LIN {X 0,Y 517.337,Z 394.066,A -85,B 0,C 180,E1 -4968.019,E2 -4968.019} C_VEL
LIN {X 0,Y 517.611,Z 384.123,A -85,B 0,C 180,E1 -4969.017,E2 -4969.017} C_VEL
LIN {X 0,Y 517.898,Z 374.015,A -85,B 0,C 180,E1 -4969.831,E2 -4969.831} C_VEL
LIN {X 0,Y 518.219,Z 361.881,A -85,B 0,C 180,E1 -4970.601,E2 -4970.601} C_VEL
LIN {X 0,Y 518.436,Z 350.506,A -85,B 0,C 180,E1 -4971.157,E2 -4971.157} C_VEL
LIN {X 0,Y 518.274,Z 345.949,A -85,B 0,C 180,E1 -4971.343,E2 -4971.343} C_VEL
LIN {X 0,Y 516.939,Z 341.096,A -85,B 0,C 180,E1 -4971.561,E2 -4971.561} C_VEL
LIN {X 0,Y 516.912,Z 341.099,A -85,B 0,C 180,E1 -4974.927,E2 -4974.927} C_VEL
LIN {X 0,Y 516.926,Z 341.098,A -85,B 0,C 180,E1 -4977.904,E2 -4977.904} C_VEL
LIN {X 0,Y 516.894,Z 341.103,A -85,B 0,C 180,E1 -4980.203,E2 -4980.203} C_VEL
LIN {X 0,Y 516.898,Z 341.101,A -85,B 0,C 180,E1 -4982.946,E2 -4982.946} C_VEL
LIN {X 0,Y 516.872,Z 341.104,A -85,B 0,C 180,E1 -4985.78,E2 -4985.78} C_VEL
LIN {X 0,Y 516.881,Z 341.103,A -85,B 0,C 180,E1 -4988.715,E2 -4988.715} C_VEL
LIN {X 0,Y 516.915,Z 341.097,A -85,B 0,C 180,E1 -4991.774,E2 -4991.774} C_VEL
LIN {X 0,Y 516.923,Z 341.097,A -85,B 0,C 180,E1 -4995.009,E2 -4995.009} C_VEL
LIN {X 0,Y 516.923,Z 341.099,A -85,B 0,C 180,E1 -4998.397,E2 -4998.397} C_VEL
LIN {X 0,Y 516.906,Z 341.1,A -85,B 0,C 180,E1 -5001.286,E2 -5001.286} C_VEL
LIN {X 0,Y 516.891,Z 341.1,A -85,B 0,C 180,E1 -5004.221,E2 -5004.221} C_VEL
LIN {X 0,Y 516.898,Z 341.099,A -85,B 0,C 180,E1 -5007.053,E2 -5007.053} C_VEL
LIN {X 0,Y 516.901,Z 341.087,A -85,B 0,C 180,E1 -5009.796,E2 -5009.796} C_VEL
LIN {X 0,Y 516.929,Z 341.095,A -85,B 0,C 180,E1 -5012.467,E2 -5012.467} C_VEL
LIN {X 0,Y 516.911,Z 341.098,A -85,B 0,C 180,E1 -5015.072,E2 -5015.072} C_VEL
LIN {X 0,Y 516.886,Z 341.103,A -85,B 0,C 180,E1 -5018.462,E2 -5018.462} C_VEL
LIN {X 0,Y 516.904,Z 341.098,A -85,B 0,C 180,E1 -5020.955,E2 -5020.955} C_VEL
LIN {X 0,Y 516.916,Z 341.098,A -85,B 0,C 180,E1 -5023.41,E2 -5023.41} C_VEL
LIN {X 0,Y 516.905,Z 341.099,A -85,B 0,C 180,E1 -5025.834,E2 -5025.834} C_VEL
LIN {X 0,Y 517.002,Z 341.088,A -85,B 0,C 180,E1 -5028.234,E2 -5028.234} C_VEL
LIN {X 0,Y 516.97,Z 341.092,A -85,B 0,C 180,E1 -5031.399,E2 -5031.399} C_VEL
LIN {X 0,Y 517.008,Z 341.083,A -85,B 0,C 180,E1 -5033.757,E2 -5033.757} C_VEL
LIN {X 0,Y 517.082,Z 341.077,A -85,B 0,C 180,E1 -5037.663,E2 -5037.663} C_VEL
LIN {X 0,Y 517.093,Z 341.074,A -85,B 0,C 180,E1 -5040.779,E2 -5040.779} C_VEL
LIN {X 0,Y 517.013,Z 341.087,A -85,B 0,C 180,E1 -5043.117,E2 -5043.117} C_VEL
LIN {X 0,Y 517.008,Z 341.086,A -85,B 0,C 180,E1 -5046.243,E2 -5046.243} C_VEL
LIN {X 0,Y 516.952,Z 341.091,A -85,B 0,C 180,E1 -5049.389,E2 -5049.389} C_VEL
LIN {X 0,Y 516.949,Z 341.093,A -85,B 0,C 180,E1 -5051.807,E2 -5051.807} C_VEL
LIN {X 0,Y 516.941,Z 341.095,A -85,B 0,C 180,E1 -5055.147,E2 -5055.147} C_VEL
LIN {X 0,Y 516.923,Z 341.097,A -85,B 0,C 180,E1 -5058.222,E2 -5058.222} C_VEL
LIN {X 0,Y 516.909,Z 341.097,A -85,B 0,C 180,E1 -5060.702,E2 -5060.702} C_VEL
LIN {X 0,Y 516.908,Z 341.099,A -85,B 0,C 180,E1 -5064.072,E2 -5064.072} C_VEL
LIN {X 0,Y 516.927,Z 341.097,A -85,B 0,C 180,E1 -5066.658,E2 -5066.658} C_VEL
LIN {X 0,Y 516.922,Z 341.098,A -85,B 0,C 180,E1 -5069.527,E2 -5069.527} C_VEL
LIN {X 0,Y 516.899,Z 341.1,A -85,B 0,C 180,E1 -5072.545,E2 -5072.545} C_VEL
LIN {X 0,Y 516.882,Z 341.102,A -85,B 0,C 180,E1 -5075.333,E2 -5075.333} C_VEL
LIN {X 0,Y 516.884,Z 341.102,A -85,B 0,C 180,E1 -5077.944,E2 -5077.944} C_VEL
LIN {X 0,Y 516.903,Z 341.099,A -85,B 0,C 180,E1 -5080.74,E2 -5080.74} C_VEL
LIN {X 0,Y 516.881,Z 341.102,A -85,B 0,C 180,E1 -5083.903,E2 -5083.903} C_VEL
LIN {X 0,Y 516.882,Z 341.101,A -85,B 0,C 180,E1 -5086.107,E2 -5086.107} C_VEL
LIN {X 0,Y 516.907,Z 341.102,A -85,B 0,C 180,E1 -5089.261,E2 -5089.261} C_VEL
LIN {X 0,Y 516.925,Z 341.244,A -85,B 0,C 180,E1 -5091.538,E2 -5091.538} C_VEL
LIN {X 0,Y 518.509,Z 349.549,A -85,B 0,C 180,E1 -5093.871,E2 -5093.871} C_VEL
LIN {X 0,Y 518.338,Z 357.102,A -85,B 0,C 180,E1 -5095.8,E2 -5095.8} C_VEL
LIN {X 0,Y 517.884,Z 371.915,A -85,B 0,C 180,E1 -5099.41,E2 -5099.41} C_VEL
LIN {X 0,Y 517.599,Z 385.199,A -85,B 0,C 180,E1 -5102.507,E2 -5102.507} C_VEL
LIN {X 0,Y 517.364,Z 398.58,A -85,B 0,C 180,E1 -5105.526,E2 -5105.526} C_VEL
LIN {X 0,Y 517.164,Z 411.994,A -85,B 0,C 180,E1 -5108.475,E2 -5108.475} C_VEL
LIN {X 0,Y 516.997,Z 423.426,A -85,B 0,C 180,E1 -5110.959,E2 -5110.959} C_VEL
LIN {X 0,Y 516.858,Z 435.03,A -85,B 0,C 180,E1 -5113.409,E2 -5113.409} C_VEL
LIN {X 0,Y 516.733,Z 447.489,A -85,B 0,C 180,E1 -5116.056,E2 -5116.056} C_VEL
LIN {X 0,Y 518.309,Z 459.336,A -85,B 0,C 180,E1 -5116.349,E2 -5116.349} C_VEL
LIN {X 0,Y 518.198,Z 472.484,A -85,B 0,C 180,E1 -5116.77,E2 -5116.77} C_VEL
LIN {X 0,Y 517.966,Z 483.611,A -85,B 0,C 180,E1 -5117.263,E2 -5117.263} C_VEL
LIN {X 0,Y 517.668,Z 495.877,A -85,B 0,C 180,E1 -5117.972,E2 -5117.972} C_VEL
LIN {X 0,Y 517.351,Z 507.545,A -85,B 0,C 180,E1 -5118.839,E2 -5118.839} C_VEL
LIN {X 0,Y 517.042,Z 518.18,A -85,B 0,C 180,E1 -5119.823,E2 -5119.823} C_VEL
LIN {X 0,Y 516.815,Z 526.807,A -85,B 0,C 180,E1 -5120.806,E2 -5120.806} C_VEL
LIN {X 0,Y 516.616,Z 535.236,A -85,B 0,C 180,E1 -5121.985,E2 -5121.985} C_VEL
LIN {X 0,Y 516.48,Z 542.24,A -85,B 0,C 180,E1 -5123.2,E2 -5123.2} C_VEL
LIN {X 0,Y 516.405,Z 548.283,A -85,B 0,C 180,E1 -5124.534,E2 -5124.534} C_VEL
LIN {X 0,Y 516.36,Z 552.34,A -85,B 0,C 180,E1 -5125.707,E2 -5125.707} C_VEL
LIN {X 0,Y 516.282,Z 555.331,A -85,B 0,C 180,E1 -5126.879,E2 -5126.879} C_VEL
LIN {X 0,Y 516.261,Z 556.758,A -85,B 0,C 180,E1 -5127.66,E2 -5127.66} C_VEL
LIN {X 0,Y 516.161,Z 558.388,A -85,B 0,C 180,E1 -5129.22,E2 -5129.22} C_VEL
LIN {X 0,Y 516.158,Z 558.609,A -85,B 0,C 180,E1 -5130.001,E2 -5130.001} C_VEL
LIN {X 0,Y 516.161,Z 558.388,A -85,B 0,C 180,E1 -5130.781,E2 -5130.781} C_VEL
LIN {X 0,Y 516.261,Z 556.761,A -85,B 0,C 180,E1 -5132.341,E2 -5132.341} C_VEL
LIN {X 0,Y 516.282,Z 555.335,A -85,B 0,C 180,E1 -5133.122,E2 -5133.122} C_VEL
LIN {X 0,Y 516.343,Z 552.34,A -85,B 0,C 180,E1 -5134.294,E2 -5134.294} C_VEL
LIN {X 0,Y 516.405,Z 548.284,A -85,B 0,C 180,E1 -5135.467,E2 -5135.467} C_VEL
LIN {X 0,Y 516.481,Z 542.255,A -85,B 0,C 180,E1 -5136.799,E2 -5136.799} C_VEL
LIN {X 0,Y 516.617,Z 535.245,A -85,B 0,C 180,E1 -5138.016,E2 -5138.016} C_VEL
LIN {X 0,Y 516.816,Z 526.82,A -85,B 0,C 180,E1 -5139.195,E2 -5139.195} C_VEL
LIN {X 0,Y 517.038,Z 518.196,A -85,B 0,C 180,E1 -5140.179,E2 -5140.179} C_VEL
LIN {X 0,Y 517.39,Z 507.571,A -85,B 0,C 180,E1 -5141.162,E2 -5141.162} C_VEL
LIN {X 0,Y 517.627,Z 496.24,A -85,B 0,C 180,E1 -5142.007,E2 -5142.007} C_VEL
LIN {X 0,Y 517.95,Z 485.582,A -85,B 0,C 180,E1 -5142.639,E2 -5142.639} C_VEL
LIN {X 0,Y 518.174,Z 473.805,A -85,B 0,C 180,E1 -5143.182,E2 -5143.182} C_VEL
LIN {X 0,Y 518.435,Z 460.279,A -85,B 0,C 180,E1 -5143.624,E2 -5143.624} C_VEL
LIN {X 0,Y 516.87,Z 449.371,A -85,B 0,C 180,E1 -5143.898,E2 -5143.898} C_VEL
LIN {X 0,Y 516.731,Z 447.432,A -85,B 0,C 180,E1 -5143.971,E2 -5143.971} C_VEL
LIN {X 0,Y 516.937,Z 433.234,A -85,B 0,C 180,E1 -5146.996,E2 -5146.996} C_VEL
LIN {X 0,Y 517.111,Z 417.675,A -85,B 0,C 180,E1 -5150.319,E2 -5150.319} C_VEL
LIN {X 0,Y 517.307,Z 404.507,A -85,B 0,C 180,E1 -5153.203,E2 -5153.203} C_VEL
LIN {X 0,Y 517.52,Z 390.545,A -85,B 0,C 180,E1 -5156.325,E2 -5156.325} C_VEL
LIN {X 0,Y 517.743,Z 377.723,A -85,B 0,C 180,E1 -5159.254,E2 -5159.254} C_VEL
LIN {X 0,Y 518.003,Z 366.207,A -85,B 0,C 180,E1 -5161.947,E2 -5161.947} C_VEL
LIN {X 0,Y 518.417,Z 352.975,A -85,B 0,C 180,E1 -5165.141,E2 -5165.141} C_VEL
LIN {X 0,Y 518.322,Z 348.977,A -85,B 0,C 180,E1 -5166.145,E2 -5166.145} C_VEL
LIN {X 0,Y 516.879,Z 341.103,A -85,B 0,C 180,E1 -5168.305,E2 -5168.305} C_VEL
LIN {X 0,Y 516.921,Z 341.098,A -85,B 0,C 180,E1 -5171.602,E2 -5171.602} C_VEL
LIN {X 0,Y 516.928,Z 341.098,A -85,B 0,C 180,E1 -5175.01,E2 -5175.01} C_VEL
LIN {X 0,Y 516.92,Z 341.098,A -85,B 0,C 180,E1 -5178.399,E2 -5178.399} C_VEL
LIN {X 0,Y 516.888,Z 341.101,A -85,B 0,C 180,E1 -5181.285,E2 -5181.285} C_VEL
LIN {X 0,Y 516.876,Z 341.103,A -85,B 0,C 180,E1 -5184.22,E2 -5184.22} C_VEL
LIN {X 0,Y 516.902,Z 341.1,A -85,B 0,C 180,E1 -5187.054,E2 -5187.054} C_VEL
LIN {X 0,Y 516.898,Z 341.1,A -85,B 0,C 180,E1 -5189.797,E2 -5189.797} C_VEL
LIN {X 0,Y 516.931,Z 341.095,A -85,B 0,C 180,E1 -5192.468,E2 -5192.468} C_VEL
LIN {X 0,Y 516.916,Z 341.099,A -85,B 0,C 180,E1 -5195.072,E2 -5195.072} C_VEL
LIN {X 0,Y 516.876,Z 341.102,A -85,B 0,C 180,E1 -5197.622,E2 -5197.622} C_VEL
LIN {X 0,Y 516.937,Z 341.095,A -85,B 0,C 180,E1 -5200.13,E2 -5200.13} C_VEL
LIN {X 0,Y 516.913,Z 341.098,A -85,B 0,C 180,E1 -5202.596,E2 -5202.596} C_VEL
LIN {X 0,Y 516.948,Z 341.094,A -85,B 0,C 180,E1 -5205.03,E2 -5205.03} C_VEL
LIN {X 0,Y 516.972,Z 341.091,A -85,B 0,C 180,E1 -5208.234,E2 -5208.234} C_VEL
LIN {X 0,Y 516.972,Z 341.089,A -85,B 0,C 180,E1 -5211.4,E2 -5211.4} C_VEL
LIN {X 0,Y 517.016,Z 341.084,A -85,B 0,C 180,E1 -5213.757,E2 -5213.757} C_VEL
LIN {X 0,Y 517.087,Z 341.077,A -85,B 0,C 180,E1 -5217.663,E2 -5217.663} C_VEL
LIN {X 0,Y 517.101,Z 341.075,A -85,B 0,C 180,E1 -5220.779,E2 -5220.779} C_VEL
LIN {X 0,Y 517.018,Z 341.085,A -85,B 0,C 180,E1 -5223.117,E2 -5223.117} C_VEL
LIN {X 0,Y 517.015,Z 341.086,A -85,B 0,C 180,E1 -5226.243,E2 -5226.243} C_VEL
LIN {X 0,Y 516.961,Z 341.091,A -85,B 0,C 180,E1 -5229.389,E2 -5229.389} C_VEL
LIN {X 0,Y 516.959,Z 341.092,A -85,B 0,C 180,E1 -5231.807,E2 -5231.807} C_VEL
LIN {X 0,Y 516.951,Z 341.092,A -85,B 0,C 180,E1 -5235.147,E2 -5235.147} C_VEL
LIN {X 0,Y 516.932,Z 341.095,A -85,B 0,C 180,E1 -5238.222,E2 -5238.222} C_VEL
LIN {X 0,Y 516.919,Z 341.096,A -85,B 0,C 180,E1 -5240.702,E2 -5240.702} C_VEL
LIN {X 0,Y 516.918,Z 341.097,A -85,B 0,C 180,E1 -5244.072,E2 -5244.072} C_VEL
LIN {X 0,Y 516.932,Z 341.096,A -85,B 0,C 180,E1 -5246.658,E2 -5246.658} C_VEL
LIN {X 0,Y 516.917,Z 341.098,A -85,B 0,C 180,E1 -5249.524,E2 -5249.524} C_VEL
LIN {X 0,Y 516.904,Z 341.099,A -85,B 0,C 180,E1 -5252.544,E2 -5252.544} C_VEL
LIN {X 0,Y 516.873,Z 341.103,A -85,B 0,C 180,E1 -5255.33,E2 -5255.33} C_VEL
LIN {X 0,Y 516.888,Z 341.102,A -85,B 0,C 180,E1 -5257.943,E2 -5257.943} C_VEL
LIN {X 0,Y 516.891,Z 341.1,A -85,B 0,C 180,E1 -5260.741,E2 -5260.741} C_VEL
LIN {X 0,Y 516.889,Z 341.101,A -85,B 0,C 180,E1 -5262.831,E2 -5262.831} C_VEL
LIN {X 0,Y 516.93,Z 341.097,A -85,B 0,C 180,E1 -5265.01,E2 -5265.01} C_VEL
LIN {X 0,Y 516.923,Z 341.097,A -85,B 0,C 180,E1 -5268.398,E2 -5268.398} C_VEL
LIN {X 0,Y 516.888,Z 341.101,A -85,B 0,C 180,E1 -5270.301,E2 -5270.301} C_VEL
LIN {X 0,Y 516.213,Z 341.185,A -85,B 0,C 180,E1 -5270.951,E2 -5270.951} C_VEL
LIN {X 0,Y 513.355,Z 341.544,A -85,B 0,C 180,E1 -5272.006,E2 -5272.006} C_VEL
LIN {X 0,Y 510.94,Z 341.846,A -85,B 0,C 180,E1 -5272.857,E2 -5272.857} C_VEL
LIN {X 0,Y 509.9,Z 341.974,A -85,B 0,C 180,E1 -5273.513,E2 -5273.513} C_VEL
LIN {X 0,Y 509.813,Z 341.983,A -85,B 0,C 180,E1 -5273.736,E2 -5273.736} C_VEL
LIN {X 0,Y 509.866,Z 341.975,A -85,B 0,C 180,E1 -5276.539,E2 -5276.539} C_VEL
LIN {X 0,Y 509.85,Z 341.979,A -85,B 0,C 180,E1 -5279.334,E2 -5279.334} C_VEL
LIN {X 0,Y 509.897,Z 341.97,A -85,B 0,C 180,E1 -5282.054,E2 -5282.054} C_VEL
LIN {X 0,Y 509.884,Z 341.974,A -85,B 0,C 180,E1 -5284.704,E2 -5284.704} C_VEL
LIN {X 0,Y 509.834,Z 341.979,A -85,B 0,C 180,E1 -5287.458,E2 -5287.458} C_VEL
LIN {X 0,Y 509.924,Z 341.967,A -85,B 0,C 180,E1 -5289.844,E2 -5289.844} C_VEL
LIN {X 0,Y 509.889,Z 341.972,A -85,B 0,C 180,E1 -5293.174,E2 -5293.174} C_VEL
LIN {X 0,Y 509.871,Z 341.973,A -85,B 0,C 180,E1 -5295.634,E2 -5295.634} C_VEL
LIN {X 0,Y 509.921,Z 341.969,A -85,B 0,C 180,E1 -5298.874,E2 -5298.874} C_VEL
LIN {X 0,Y 509.959,Z 341.964,A -85,B 0,C 180,E1 -5302.078,E2 -5302.078} C_VEL
LIN {X 0,Y 509.974,Z 341.963,A -85,B 0,C 180,E1 -5304.34,E2 -5304.34} C_VEL
LIN {X 0,Y 511.619,Z 348.18,A -85,B 0,C 180,E1 -5304.63,E2 -5304.63} C_VEL
LIN {X 0,Y 511.412,Z 359.998,A -85,B 0,C 180,E1 -5305.171,E2 -5305.171} C_VEL
LIN {X 0,Y 511.143,Z 371.42,A -85,B 0,C 180,E1 -5305.86,E2 -5305.86} C_VEL
LIN {X 0,Y 510.795,Z 382.869,A -85,B 0,C 180,E1 -5306.746,E2 -5306.746} C_VEL
LIN {X 0,Y 510.5,Z 392.107,A -85,B 0,C 180,E1 -5307.632,E2 -5307.632} C_VEL
LIN {X 0,Y 510.193,Z 400.557,A -85,B 0,C 180,E1 -5308.618,E2 -5308.618} C_VEL
LIN {X 0,Y 509.931,Z 408.768,A -85,B 0,C 180,E1 -5309.802,E2 -5309.802} C_VEL
LIN {X 0,Y 509.631,Z 416.37,A -85,B 0,C 180,E1 -5311.185,E2 -5311.185} C_VEL
LIN {X 0,Y 509.497,Z 421.464,A -85,B 0,C 180,E1 -5312.371,E2 -5312.371} C_VEL
LIN {X 0,Y 509.46,Z 425.423,A -85,B 0,C 180,E1 -5313.558,E2 -5313.558} C_VEL
LIN {X 0,Y 509.347,Z 428.382,A -85,B 0,C 180,E1 -5314.748,E2 -5314.748} C_VEL
LIN {X 0,Y 509.37,Z 429.832,A -85,B 0,C 180,E1 -5315.542,E2 -5315.542} C_VEL
LIN {X 0,Y 509.331,Z 431.496,A -85,B 0,C 180,E1 -5317.133,E2 -5317.133} C_VEL
LIN {X 0,Y 509.334,Z 431.764,A -85,B 0,C 180,E1 -5317.931,E2 -5317.931} C_VEL
LIN {X 0,Y 509.303,Z 431.64,A -85,B 0,C 180,E1 -5318.73,E2 -5318.73} C_VEL
LIN {X 0,Y 509.29,Z 430.153,A -85,B 0,C 180,E1 -5320.334,E2 -5320.334} C_VEL
LIN {X 0,Y 509.393,Z 427.838,A -85,B 0,C 180,E1 -5321.598,E2 -5321.598} C_VEL
LIN {X 0,Y 509.441,Z 424.792,A -85,B 0,C 180,E1 -5322.751,E2 -5322.751} C_VEL
LIN {X 0,Y 509.555,Z 420.523,A -85,B 0,C 180,E1 -5323.967,E2 -5323.967} C_VEL
LIN {X 0,Y 509.743,Z 415.022,A -85,B 0,C 180,E1 -5325.186,E2 -5325.186} C_VEL
LIN {X 0,Y 509.929,Z 408.09,A -85,B 0,C 180,E1 -5326.411,E2 -5326.411} C_VEL
LIN {X 0,Y 510.241,Z 399.294,A -85,B 0,C 180,E1 -5327.639,E2 -5327.639} C_VEL
LIN {X 0,Y 510.571,Z 390.201,A -85,B 0,C 180,E1 -5328.664,E2 -5328.664} C_VEL
LIN {X 0,Y 510.846,Z 380.073,A -85,B 0,C 180,E1 -5329.593,E2 -5329.593} C_VEL
LIN {X 0,Y 511.197,Z 369.49,A -85,B 0,C 180,E1 -5330.364,E2 -5330.364} C_VEL
LIN {X 0,Y 511.481,Z 357.788,A -85,B 0,C 180,E1 -5331.036,E2 -5331.036} C_VEL
LIN {X 0,Y 511.617,Z 348.497,A -85,B 0,C 180,E1 -5331.453,E2 -5331.453} C_VEL
LIN {X 0,Y 509.877,Z 341.975,A -85,B 0,C 180,E1 -5331.768,E2 -5331.768} C_VEL
LIN {X 0,Y 509.879,Z 341.975,A -85,B 0,C 180,E1 -5335.295,E2 -5335.295} C_VEL
LIN {X 0,Y 509.898,Z 341.973,A -85,B 0,C 180,E1 -5338.1,E2 -5338.1} C_VEL
LIN {X 0,Y 509.848,Z 341.978,A -85,B 0,C 180,E1 -5341.279,E2 -5341.279} C_VEL
LIN {X 0,Y 509.858,Z 341.976,A -85,B 0,C 180,E1 -5344.202,E2 -5344.202} C_VEL
LIN {X 0,Y 509.817,Z 341.984,A -85,B 0,C 180,E1 -5347.34,E2 -5347.34} C_VEL
LIN {X 0,Y 509.839,Z 341.98,A -85,B 0,C 180,E1 -5350.381,E2 -5350.381} C_VEL
LIN {X 0,Y 509.84,Z 341.979,A -85,B 0,C 180,E1 -5353.064,E2 -5353.064} C_VEL
LIN {X 0,Y 509.831,Z 341.981,A -85,B 0,C 180,E1 -5355.792,E2 -5355.792} C_VEL
LIN {X 0,Y 509.865,Z 341.978,A -85,B 0,C 180,E1 -5358.575,E2 -5358.575} C_VEL
LIN {X 0,Y 509.859,Z 341.978,A -85,B 0,C 180,E1 -5361.662,E2 -5361.662} C_VEL
LIN {X 0,Y 509.847,Z 341.979,A -85,B 0,C 180,E1 -5364.623,E2 -5364.623} C_VEL
LIN {X 0,Y 509.866,Z 341.974,A -85,B 0,C 180,E1 -5367.481,E2 -5367.481} C_VEL
LIN {X 0,Y 509.88,Z 341.962,A -85,B 0,C 180,E1 -5370.268,E2 -5370.268} C_VEL
LIN {X 0,Y 509.886,Z 341.971,A -85,B 0,C 180,E1 -5372.944,E2 -5372.944} C_VEL
LIN {X 0,Y 509.869,Z 341.974,A -85,B 0,C 180,E1 -5375.574,E2 -5375.574} C_VEL
LIN {X 0,Y 509.821,Z 341.98,A -85,B 0,C 180,E1 -5378.148,E2 -5378.148} C_VEL
LIN {X 0,Y 509.864,Z 341.975,A -85,B 0,C 180,E1 -5380.681,E2 -5380.681} C_VEL
LIN {X 0,Y 509.886,Z 341.971,A -85,B 0,C 180,E1 -5383.175,E2 -5383.175} C_VEL
LIN {X 0,Y 509.872,Z 341.975,A -85,B 0,C 180,E1 -5385.634,E2 -5385.634} C_VEL
LIN {X 0,Y 509.929,Z 341.968,A -85,B 0,C 180,E1 -5388.875,E2 -5388.875} C_VEL
LIN {X 0,Y 509.95,Z 341.966,A -85,B 0,C 180,E1 -5392.078,E2 -5392.078} C_VEL
LIN {X 0,Y 509.981,Z 341.959,A -85,B 0,C 180,E1 -5394.464,E2 -5394.464} C_VEL
LIN {X 0,Y 510.053,Z 341.952,A -85,B 0,C 180,E1 -5397.631,E2 -5397.631} C_VEL
LIN {X 0,Y 510.063,Z 341.949,A -85,B 0,C 180,E1 -5400.789,E2 -5400.789} C_VEL
LIN {X 0,Y 509.955,Z 341.966,A -85,B 0,C 180,E1 -5403.16,E2 -5403.16} C_VEL
LIN {X 0,Y 509.976,Z 341.963,A -85,B 0,C 180,E1 -5406.329,E2 -5406.329} C_VEL
LIN {X 0,Y 509.914,Z 341.969,A -85,B 0,C 180,E1 -5408.72,E2 -5408.72} C_VEL
LIN {X 0,Y 509.901,Z 341.971,A -85,B 0,C 180,E1 -5411.932,E2 -5411.932} C_VEL
LIN {X 0,Y 509.89,Z 341.974,A -85,B 0,C 180,E1 -5415.242,E2 -5415.242} C_VEL
LIN {X 0,Y 509.885,Z 341.972,A -85,B 0,C 180,E1 -5418.001,E2 -5418.001} C_VEL
LIN {X 0,Y 509.847,Z 341.977,A -85,B 0,C 180,E1 -5421.002,E2 -5421.002} C_VEL
LIN {X 0,Y 509.834,Z 341.979,A -85,B 0,C 180,E1 -5423.563,E2 -5423.563} C_VEL
LIN {X 0,Y 509.911,Z 341.972,A -85,B 0,C 180,E1 -5426.379,E2 -5426.379} C_VEL
LIN {X 0,Y 509.883,Z 341.975,A -85,B 0,C 180,E1 -5428.844,E2 -5428.844} C_VEL
LIN {X 0,Y 509.824,Z 341.982,A -85,B 0,C 180,E1 -5431.59,E2 -5431.59} C_VEL
LIN {X 0,Y 509.852,Z 341.978,A -85,B 0,C 180,E1 -5434.413,E2 -5434.413} C_VEL
LIN {X 0,Y 509.821,Z 341.982,A -85,B 0,C 180,E1 -5437.341,E2 -5437.341} C_VEL
LIN {X 0,Y 509.86,Z 341.977,A -85,B 0,C 180,E1 -5440.38,E2 -5440.38} C_VEL
LIN {X 0,Y 509.838,Z 341.981,A -85,B 0,C 180,E1 -5443.065,E2 -5443.065} C_VEL
LIN {X 0,Y 509.83,Z 341.981,A -85,B 0,C 180,E1 -5445.793,E2 -5445.793} C_VEL
LIN {X 0,Y 509.87,Z 341.977,A -85,B 0,C 180,E1 -5448.577,E2 -5448.577} C_VEL
LIN {X 0,Y 509.906,Z 342.094,A -85,B 0,C 180,E1 -5451.258,E2 -5451.258} C_VEL
LIN {X 0,Y 511.562,Z 350.947,A -85,B 0,C 180,E1 -5453.791,E2 -5453.791} C_VEL
LIN {X 0,Y 511.394,Z 358.315,A -85,B 0,C 180,E1 -5455.706,E2 -5455.706} C_VEL
LIN {X 0,Y 510.939,Z 371.404,A -85,B 0,C 180,E1 -5458.959,E2 -5458.959} C_VEL
LIN {X 0,Y 510.599,Z 384.561,A -85,B 0,C 180,E1 -5462.097,E2 -5462.097} C_VEL
LIN {X 0,Y 510.365,Z 397.528,A -85,B 0,C 180,E1 -5465.088,E2 -5465.088} C_VEL
LIN {X 0,Y 510.12,Z 411.233,A -85,B 0,C 180,E1 -5468.163,E2 -5468.163} C_VEL
LIN {X 0,Y 509.933,Z 422.681,A -85,B 0,C 180,E1 -5470.685,E2 -5470.685} C_VEL
LIN {X 0,Y 509.793,Z 434.11,A -85,B 0,C 180,E1 -5473.172,E2 -5473.172} C_VEL
LIN {X 0,Y 509.66,Z 446.577,A -85,B 0,C 180,E1 -5475.858,E2 -5475.858} C_VEL
LIN {X 0,Y 511.033,Z 457.931,A -85,B 0,C 180,E1 -5476.138,E2 -5476.138} C_VEL
LIN {X 0,Y 511.475,Z 462.135,A -85,B 0,C 180,E1 -5476.264,E2 -5476.264} C_VEL
LIN {X 0,Y 511.177,Z 475.257,A -85,B 0,C 180,E1 -5476.737,E2 -5476.737} C_VEL
LIN {X 0,Y 510.84,Z 487.929,A -85,B 0,C 180,E1 -5477.369,E2 -5477.369} C_VEL
LIN {X 0,Y 510.567,Z 499.026,A -85,B 0,C 180,E1 -5478.085,E2 -5478.085} C_VEL
LIN {X 0,Y 510.21,Z 510.079,A -85,B 0,C 180,E1 -5478.982,E2 -5478.982} C_VEL
LIN {X 0,Y 509.927,Z 519.109,A -85,B 0,C 180,E1 -5479.88,E2 -5479.88} C_VEL
LIN {X 0,Y 509.68,Z 528.943,A -85,B 0,C 180,E1 -5481.076,E2 -5481.076} C_VEL
LIN {X 0,Y 509.512,Z 536.792,A -85,B 0,C 180,E1 -5482.272,E2 -5482.272} C_VEL
LIN {X 0,Y 509.341,Z 544.029,A -85,B 0,C 180,E1 -5483.663,E2 -5483.663} C_VEL
LIN {X 0,Y 509.255,Z 548.853,A -85,B 0,C 180,E1 -5484.854,E2 -5484.854} C_VEL
LIN {X 0,Y 509.303,Z 552.555,A -85,B 0,C 180,E1 -5486.044,E2 -5486.044} C_VEL
LIN {X 0,Y 509.232,Z 554.454,A -85,B 0,C 180,E1 -5486.836,E2 -5486.836} C_VEL
LIN {X 0,Y 509.206,Z 555.882,A -85,B 0,C 180,E1 -5487.628,E2 -5487.628} C_VEL
LIN {X 0,Y 509.114,Z 557.515,A -85,B 0,C 180,E1 -5489.21,E2 -5489.21} C_VEL
LIN {X 0,Y 509.112,Z 557.738,A -85,B 0,C 180,E1 -5490.001,E2 -5490.001} C_VEL
LIN {X 0,Y 509.114,Z 557.517,A -85,B 0,C 180,E1 -5490.792,E2 -5490.792} C_VEL
LIN {X 0,Y 509.205,Z 555.89,A -85,B 0,C 180,E1 -5492.374,E2 -5492.374} C_VEL
LIN {X 0,Y 509.232,Z 554.465,A -85,B 0,C 180,E1 -5493.165,E2 -5493.165} C_VEL
LIN {X 0,Y 509.269,Z 551.466,A -85,B 0,C 180,E1 -5494.354,E2 -5494.354} C_VEL
LIN {X 0,Y 509.344,Z 547.412,A -85,B 0,C 180,E1 -5495.543,E2 -5495.543} C_VEL
LIN {X 0,Y 509.403,Z 541.634,A -85,B 0,C 180,E1 -5496.845,E2 -5496.845} C_VEL
LIN {X 0,Y 509.563,Z 534.37,A -85,B 0,C 180,E1 -5498.128,E2 -5498.128} C_VEL
LIN {X 0,Y 509.759,Z 525.944,A -85,B 0,C 180,E1 -5499.323,E2 -5499.323} C_VEL
LIN {X 0,Y 510.006,Z 517.32,A -85,B 0,C 180,E1 -5500.32,E2 -5500.32} C_VEL
LIN {X 0,Y 510.353,Z 506.691,A -85,B 0,C 180,E1 -5501.317,E2 -5501.317} C_VEL
LIN {X 0,Y 510.616,Z 495.361,A -85,B 0,C 180,E1 -5502.174,E2 -5502.174} C_VEL
LIN {X 0,Y 510.959,Z 484.704,A -85,B 0,C 180,E1 -5502.815,E2 -5502.815} C_VEL
LIN {X 0,Y 511.239,Z 472.931,A -85,B 0,C 180,E1 -5503.364,E2 -5503.364} C_VEL
LIN {X 0,Y 511.36,Z 460.306,A -85,B 0,C 180,E1 -5503.791,E2 -5503.791} C_VEL
LIN {X 0,Y 509.739,Z 448.093,A -85,B 0,C 180,E1 -5504.103,E2 -5504.103} C_VEL
LIN {X 0,Y 509.676,Z 446.545,A -85,B 0,C 180,E1 -5504.168,E2 -5504.168} C_VEL
LIN {X 0,Y 509.89,Z 430.427,A -85,B 0,C 180,E1 -5507.653,E2 -5507.653} C_VEL
LIN {X 0,Y 510.045,Z 416.632,A -85,B 0,C 180,E1 -5510.676,E2 -5510.676} C_VEL
LIN {X 0,Y 510.269,Z 403.803,A -85,B 0,C 180,E1 -5513.543,E2 -5513.543} C_VEL
LIN {X 0,Y 510.493,Z 390.743,A -85,B 0,C 180,E1 -5516.509,E2 -5516.509} C_VEL
LIN {X 0,Y 510.791,Z 377.023,A -85,B 0,C 180,E1 -5519.692,E2 -5519.692} C_VEL
LIN {X 0,Y 511.079,Z 364.376,A -85,B 0,C 180,E1 -5522.709,E2 -5522.709} C_VEL
LIN {X 0,Y 511.487,Z 352.891,A -85,B 0,C 180,E1 -5525.539,E2 -5525.539} C_VEL
LIN {X 0,Y 511.122,Z 348.652,A -85,B 0,C 180,E1 -5526.643,E2 -5526.643} C_VEL
LIN {X 0,Y 509.852,Z 341.979,A -85,B 0,C 180,E1 -5528.465,E2 -5528.465} C_VEL
LIN {X 0,Y 509.862,Z 341.977,A -85,B 0,C 180,E1 -5531.426,E2 -5531.426} C_VEL
LIN {X 0,Y 509.862,Z 341.978,A -85,B 0,C 180,E1 -5534.668,E2 -5534.668} C_VEL
LIN {X 0,Y 509.861,Z 341.975,A -85,B 0,C 180,E1 -5538.104,E2 -5538.104} C_VEL
LIN {X 0,Y 509.853,Z 341.978,A -85,B 0,C 180,E1 -5540.648,E2 -5540.648} C_VEL
LIN {X 0,Y 509.83,Z 341.98,A -85,B 0,C 180,E1 -5543.647,E2 -5543.647} C_VEL
LIN {X 0,Y 509.865,Z 341.977,A -85,B 0,C 180,E1 -5546.54,E2 -5546.54} C_VEL
LIN {X 0,Y 509.852,Z 341.978,A -85,B 0,C 180,E1 -5549.335,E2 -5549.335} C_VEL
LIN {X 0,Y 509.897,Z 341.972,A -85,B 0,C 180,E1 -5552.055,E2 -5552.055} C_VEL
LIN {X 0,Y 509.882,Z 341.974,A -85,B 0,C 180,E1 -5554.704,E2 -5554.704} C_VEL
LIN {X 0,Y 509.862,Z 341.976,A -85,B 0,C 180,E1 -5557.45,E2 -5557.45} C_VEL
LIN {X 0,Y 509.922,Z 341.969,A -85,B 0,C 180,E1 -5559.845,E2 -5559.845} C_VEL
LIN {X 0,Y 509.881,Z 341.974,A -85,B 0,C 180,E1 -5563.175,E2 -5563.175} C_VEL
LIN {X 0,Y 509.87,Z 341.975,A -85,B 0,C 180,E1 -5565.634,E2 -5565.634} C_VEL
LIN {X 0,Y 509.918,Z 341.969,A -85,B 0,C 180,E1 -5568.875,E2 -5568.875} C_VEL
LIN {X 0,Y 509.957,Z 341.966,A -85,B 0,C 180,E1 -5572.079,E2 -5572.079} C_VEL
LIN {X 0,Y 509.988,Z 341.961,A -85,B 0,C 180,E1 -5574.465,E2 -5574.465} C_VEL
LIN {X 0,Y 510.058,Z 341.952,A -85,B 0,C 180,E1 -5577.631,E2 -5577.631} C_VEL
LIN {X 0,Y 510.071,Z 341.951,A -85,B 0,C 180,E1 -5580.79,E2 -5580.79} C_VEL
LIN {X 0,Y 509.96,Z 341.964,A -85,B 0,C 180,E1 -5583.16,E2 -5583.16} C_VEL
LIN {X 0,Y 509.984,Z 341.962,A -85,B 0,C 180,E1 -5586.33,E2 -5586.33} C_VEL
LIN {X 0,Y 509.923,Z 341.969,A -85,B 0,C 180,E1 -5588.72,E2 -5588.72} C_VEL
LIN {X 0,Y 509.911,Z 341.971,A -85,B 0,C 180,E1 -5591.932,E2 -5591.932} C_VEL
LIN {X 0,Y 509.901,Z 341.97,A -85,B 0,C 180,E1 -5595.242,E2 -5595.242} C_VEL
LIN {X 0,Y 509.895,Z 341.973,A -85,B 0,C 180,E1 -5598.001,E2 -5598.001} C_VEL
LIN {X 0,Y 509.857,Z 341.976,A -85,B 0,C 180,E1 -5601.002,E2 -5601.002} C_VEL
LIN {X 0,Y 509.877,Z 341.975,A -85,B 0,C 180,E1 -5604.426,E2 -5604.426} C_VEL
LIN {X 0,Y 509.891,Z 341.973,A -85,B 0,C 180,E1 -5607.056,E2 -5607.056} C_VEL
LIN {X 0,Y 509.864,Z 341.976,A -85,B 0,C 180,E1 -5609.751,E2 -5609.751} C_VEL
LIN {X 0,Y 509.881,Z 341.973,A -85,B 0,C 180,E1 -5612.774,E2 -5612.774} C_VEL
LIN {X 0,Y 509.833,Z 341.981,A -85,B 0,C 180,E1 -5615.578,E2 -5615.578} C_VEL
LIN {X 0,Y 509.858,Z 341.975,A -85,B 0,C 180,E1 -5618.338,E2 -5618.338} C_VEL
LIN {X 0,Y 509.864,Z 341.978,A -85,B 0,C 180,E1 -5621.425,E2 -5621.425} C_VEL
LIN {X 0,Y 509.864,Z 341.976,A -85,B 0,C 180,E1 -5624.668,E2 -5624.668} C_VEL
LIN {X 0,Y 509.865,Z 341.976,A -85,B 0,C 180,E1 -5628.103,E2 -5628.103} C_VEL
LIN {X 0,Y 509.852,Z 341.978,A -85,B 0,C 180,E1 -5630.647,E2 -5630.647} C_VEL
LIN {X 0,Y 509.813,Z 341.983,A -85,B 0,C 180,E1 -5633.736,E2 -5633.736} C_VEL
LIN {X 0,Y 509.154,Z 342.063,A -85,B 0,C 180,E1 -5634.395,E2 -5634.395} C_VEL
LIN {X 0,Y 506.347,Z 342.414,A -85,B 0,C 180,E1 -5635.468,E2 -5635.468} C_VEL
LIN {X 0,Y 503.96,Z 342.713,A -85,B 0,C 180,E1 -5636.331,E2 -5636.331} C_VEL
LIN {X 0,Y 502.913,Z 342.843,A -85,B 0,C 180,E1 -5636.998,E2 -5636.998} C_VEL
LIN {X 0,Y 502.815,Z 342.853,A -85,B 0,C 180,E1 -5637.223,E2 -5637.223} C_VEL
LIN {X 0,Y 502.821,Z 342.852,A -85,B 0,C 180,E1 -5640.065,E2 -5640.065} C_VEL
LIN {X 0,Y 502.838,Z 342.851,A -85,B 0,C 180,E1 -5642.533,E2 -5642.533} C_VEL
LIN {X 0,Y 502.834,Z 342.851,A -85,B 0,C 180,E1 -5645.299,E2 -5645.299} C_VEL
LIN {X 0,Y 502.787,Z 342.856,A -85,B 0,C 180,E1 -5647.826,E2 -5647.826} C_VEL
LIN {X 0,Y 502.832,Z 342.852,A -85,B 0,C 180,E1 -5650.4,E2 -5650.4} C_VEL
LIN {X 0,Y 502.837,Z 342.852,A -85,B 0,C 180,E1 -5652.931,E2 -5652.931} C_VEL
LIN {X 0,Y 502.852,Z 342.848,A -85,B 0,C 180,E1 -5655.429,E2 -5655.429} C_VEL
LIN {X 0,Y 502.885,Z 342.846,A -85,B 0,C 180,E1 -5658.716,E2 -5658.716} C_VEL
LIN {X 0,Y 502.909,Z 342.843,A -85,B 0,C 180,E1 -5661.966,E2 -5661.966} C_VEL
LIN {X 0,Y 502.942,Z 342.936,A -85,B 0,C 180,E1 -5664.16,E2 -5664.16} C_VEL
LIN {X 0,Y 504.776,Z 349.338,A -85,B 0,C 180,E1 -5664.457,E2 -5664.457} C_VEL
LIN {X 0,Y 504.532,Z 361.094,A -85,B 0,C 180,E1 -5665.005,E2 -5665.005} C_VEL
LIN {X 0,Y 504.261,Z 372.444,A -85,B 0,C 180,E1 -5665.703,E2 -5665.703} C_VEL
LIN {X 0,Y 503.908,Z 382.729,A -85,B 0,C 180,E1 -5666.501,E2 -5666.501} C_VEL
LIN {X 0,Y 503.61,Z 392.13,A -85,B 0,C 180,E1 -5667.4,E2 -5667.4} C_VEL
LIN {X 0,Y 503.276,Z 400.72,A -85,B 0,C 180,E1 -5668.399,E2 -5668.399} C_VEL
LIN {X 0,Y 502.982,Z 409.104,A -85,B 0,C 180,E1 -5669.599,E2 -5669.599} C_VEL
LIN {X 0,Y 502.715,Z 415.815,A -85,B 0,C 180,E1 -5670.8,E2 -5670.8} C_VEL
LIN {X 0,Y 502.518,Z 421.198,A -85,B 0,C 180,E1 -5672.003,E2 -5672.003} C_VEL
LIN {X 0,Y 502.437,Z 425.42,A -85,B 0,C 180,E1 -5673.207,E2 -5673.207} C_VEL
LIN {X 0,Y 502.357,Z 427.666,A -85,B 0,C 180,E1 -5674.011,E2 -5674.011} C_VEL
LIN {X 0,Y 502.323,Z 429.49,A -85,B 0,C 180,E1 -5674.815,E2 -5674.815} C_VEL
LIN {X 0,Y 502.331,Z 430.855,A -85,B 0,C 180,E1 -5675.62,E2 -5675.62} C_VEL
LIN {X 0,Y 502.302,Z 432.432,A -85,B 0,C 180,E1 -5677.234,E2 -5677.234} C_VEL
LIN {X 0,Y 502.291,Z 432.652,A -85,B 0,C 180,E1 -5678.043,E2 -5678.043} C_VEL
LIN {X 0,Y 502.257,Z 431.851,A -85,B 0,C 180,E1 -5679.666,E2 -5679.666} C_VEL
LIN {X 0,Y 502.275,Z 430.871,A -85,B 0,C 180,E1 -5680.48,E2 -5680.48} C_VEL
LIN {X 0,Y 502.379,Z 428.626,A -85,B 0,C 180,E1 -5681.687,E2 -5681.687} C_VEL
LIN {X 0,Y 502.449,Z 425.322,A -85,B 0,C 180,E1 -5682.932,E2 -5682.932} C_VEL
LIN {X 0,Y 502.584,Z 420.948,A -85,B 0,C 180,E1 -5684.164,E2 -5684.164} C_VEL
LIN {X 0,Y 502.786,Z 415.333,A -85,B 0,C 180,E1 -5685.401,E2 -5685.401} C_VEL
LIN {X 0,Y 502.988,Z 408.213,A -85,B 0,C 180,E1 -5686.644,E2 -5686.644} C_VEL
LIN {X 0,Y 503.327,Z 399.251,A -85,B 0,C 180,E1 -5687.889,E2 -5687.889} C_VEL
LIN {X 0,Y 503.666,Z 389.956,A -85,B 0,C 180,E1 -5688.93,E2 -5688.93} C_VEL
LIN {X 0,Y 504.014,Z 379.479,A -85,B 0,C 180,E1 -5689.869,E2 -5689.869} C_VEL
LIN {X 0,Y 504.387,Z 367.971,A -85,B 0,C 180,E1 -5690.69,E2 -5690.69} C_VEL
LIN {X 0,Y 504.658,Z 356.332,A -85,B 0,C 180,E1 -5691.335,E2 -5691.335} C_VEL
LIN {X 0,Y 504.577,Z 348.988,A -85,B 0,C 180,E1 -5691.66,E2 -5691.66} C_VEL
LIN {X 0,Y 502.816,Z 342.854,A -85,B 0,C 180,E1 -5691.955,E2 -5691.955} C_VEL
LIN {X 0,Y 502.83,Z 342.853,A -85,B 0,C 180,E1 -5694.79,E2 -5694.79} C_VEL
LIN {X 0,Y 502.834,Z 342.854,A -85,B 0,C 180,E1 -5697.466,E2 -5697.466} C_VEL
LIN {X 0,Y 502.811,Z 342.857,A -85,B 0,C 180,E1 -5700.21,E2 -5700.21} C_VEL
LIN {X 0,Y 502.833,Z 342.853,A -85,B 0,C 180,E1 -5703.03,E2 -5703.03} C_VEL
LIN {X 0,Y 502.774,Z 342.86,A -85,B 0,C 180,E1 -5705.95,E2 -5705.95} C_VEL
LIN {X 0,Y 502.802,Z 342.856,A -85,B 0,C 180,E1 -5708.975,E2 -5708.975} C_VEL
LIN {X 0,Y 502.83,Z 342.851,A -85,B 0,C 180,E1 -5712.135,E2 -5712.135} C_VEL
LIN {X 0,Y 502.801,Z 342.858,A -85,B 0,C 180,E1 -5715.467,E2 -5715.467} C_VEL
LIN {X 0,Y 502.826,Z 342.854,A -85,B 0,C 180,E1 -5719.003,E2 -5719.003} C_VEL
LIN {X 0,Y 502.797,Z 342.857,A -85,B 0,C 180,E1 -5722.046,E2 -5722.046} C_VEL
LIN {X 0,Y 502.81,Z 342.855,A -85,B 0,C 180,E1 -5725.035,E2 -5725.035} C_VEL
LIN {X 0,Y 502.787,Z 342.854,A -85,B 0,C 180,E1 -5727.915,E2 -5727.915} C_VEL
LIN {X 0,Y 502.838,Z 342.843,A -85,B 0,C 180,E1 -5730.713,E2 -5730.713} C_VEL
LIN {X 0,Y 502.879,Z 342.846,A -85,B 0,C 180,E1 -5733.434,E2 -5733.434} C_VEL
LIN {X 0,Y 502.79,Z 342.855,A -85,B 0,C 180,E1 -5736.086,E2 -5736.086} C_VEL
LIN {X 0,Y 502.782,Z 342.858,A -85,B 0,C 180,E1 -5738.688,E2 -5738.688} C_VEL
LIN {X 0,Y 502.829,Z 342.852,A -85,B 0,C 180,E1 -5741.248,E2 -5741.248} C_VEL
LIN {X 0,Y 502.822,Z 342.852,A -85,B 0,C 180,E1 -5743.767,E2 -5743.767} C_VEL
LIN {X 0,Y 502.835,Z 342.853,A -85,B 0,C 180,E1 -5746.255,E2 -5746.255} C_VEL
LIN {X 0,Y 502.9,Z 342.843,A -85,B 0,C 180,E1 -5748.717,E2 -5748.717} C_VEL
LIN {X 0,Y 502.9,Z 342.843,A -85,B 0,C 180,E1 -5751.966,E2 -5751.966} C_VEL
LIN {X 0,Y 502.937,Z 342.836,A -85,B 0,C 180,E1 -5754.386,E2 -5754.386} C_VEL
LIN {X 0,Y 503.023,Z 342.828,A -85,B 0,C 180,E1 -5757.598,E2 -5757.598} C_VEL
LIN {X 0,Y 503.024,Z 342.824,A -85,B 0,C 180,E1 -5760,E2 -5760} C_VEL
LIN {X 0,Y 503.022,Z 342.83,A -85,B 0,C 180,E1 -5762.402,E2 -5762.402} C_VEL
LIN {X 0,Y 502.937,Z 342.837,A -85,B 0,C 180,E1 -5765.613,E2 -5765.613} C_VEL
LIN {X 0,Y 502.899,Z 342.844,A -85,B 0,C 180,E1 -5768.033,E2 -5768.033} C_VEL
LIN {X 0,Y 502.874,Z 342.848,A -85,B 0,C 180,E1 -5771.283,E2 -5771.283} C_VEL
LIN {X 0,Y 502.842,Z 342.85,A -85,B 0,C 180,E1 -5774.571,E2 -5774.571} C_VEL
LIN {X 0,Y 502.859,Z 342.847,A -85,B 0,C 180,E1 -5777.907,E2 -5777.907} C_VEL
LIN {X 0,Y 502.825,Z 342.852,A -85,B 0,C 180,E1 -5780.536,E2 -5780.536} C_VEL
LIN {X 0,Y 502.793,Z 342.858,A -85,B 0,C 180,E1 -5783.04,E2 -5783.04} C_VEL
LIN {X 0,Y 502.839,Z 342.852,A -85,B 0,C 180,E1 -5785.676,E2 -5785.676} C_VEL
LIN {X 0,Y 502.84,Z 342.853,A -85,B 0,C 180,E1 -5788.373,E2 -5788.373} C_VEL
LIN {X 0,Y 502.795,Z 342.858,A -85,B 0,C 180,E1 -5791.5,E2 -5791.5} C_VEL
LIN {X 0,Y 502.805,Z 342.856,A -85,B 0,C 180,E1 -5794.445,E2 -5794.445} C_VEL
LIN {X 0,Y 502.782,Z 342.859,A -85,B 0,C 180,E1 -5797.179,E2 -5797.179} C_VEL
LIN {X 0,Y 502.824,Z 342.854,A -85,B 0,C 180,E1 -5800.012,E2 -5800.012} C_VEL
LIN {X 0,Y 502.827,Z 342.851,A -85,B 0,C 180,E1 -5802.203,E2 -5802.203} C_VEL
LIN {X 0,Y 502.799,Z 342.857,A -85,B 0,C 180,E1 -5805.469,E2 -5805.469} C_VEL
LIN {X 0,Y 502.838,Z 342.853,A -85,B 0,C 180,E1 -5807.866,E2 -5807.866} C_VEL
LIN {X 0,Y 502.83,Z 342.936,A -85,B 0,C 180,E1 -5810.963,E2 -5810.963} C_VEL
LIN {X 0,Y 504.572,Z 351.9,A -85,B 0,C 180,E1 -5813.585,E2 -5813.585} C_VEL
LIN {X 0,Y 504.553,Z 357.846,A -85,B 0,C 180,E1 -5815.174,E2 -5815.174} C_VEL
LIN {X 0,Y 503.993,Z 371.358,A -85,B 0,C 180,E1 -5818.608,E2 -5818.608} C_VEL
LIN {X 0,Y 503.617,Z 383.952,A -85,B 0,C 180,E1 -5821.676,E2 -5821.676} C_VEL
LIN {X 0,Y 503.348,Z 397.189,A -85,B 0,C 180,E1 -5824.796,E2 -5824.796} C_VEL
LIN {X 0,Y 503.092,Z 410.473,A -85,B 0,C 180,E1 -5827.842,E2 -5827.842} C_VEL
LIN {X 0,Y 502.885,Z 421.877,A -85,B 0,C 180,E1 -5830.403,E2 -5830.403} C_VEL
LIN {X 0,Y 502.741,Z 433.257,A -85,B 0,C 180,E1 -5832.929,E2 -5832.929} C_VEL
LIN {X 0,Y 502.565,Z 445.659,A -85,B 0,C 180,E1 -5835.654,E2 -5835.654} C_VEL
LIN {X 0,Y 504.07,Z 458.869,A -85,B 0,C 180,E1 -5835.994,E2 -5835.994} C_VEL
LIN {X 0,Y 504.509,Z 462.848,A -85,B 0,C 180,E1 -5836.122,E2 -5836.122} C_VEL
LIN {X 0,Y 504.185,Z 475.494,A -85,B 0,C 180,E1 -5836.601,E2 -5836.601} C_VEL
LIN {X 0,Y 503.813,Z 488.593,A -85,B 0,C 180,E1 -5837.281,E2 -5837.281} C_VEL
LIN {X 0,Y 503.482,Z 500.77,A -85,B 0,C 180,E1 -5838.119,E2 -5838.119} C_VEL
LIN {X 0,Y 503.131,Z 511.355,A -85,B 0,C 180,E1 -5839.029,E2 -5839.029} C_VEL
LIN {X 0,Y 502.843,Z 520.028,A -85,B 0,C 180,E1 -5839.939,E2 -5839.939} C_VEL
LIN {X 0,Y 502.601,Z 528.046,A -85,B 0,C 180,E1 -5840.95,E2 -5840.95} C_VEL
LIN {X 0,Y 502.423,Z 535.897,A -85,B 0,C 180,E1 -5842.162,E2 -5842.162} C_VEL
LIN {X 0,Y 502.274,Z 543.142,A -85,B 0,C 180,E1 -5843.573,E2 -5843.573} C_VEL
LIN {X 0,Y 502.197,Z 547.97,A -85,B 0,C 180,E1 -5844.782,E2 -5844.782} C_VEL
LIN {X 0,Y 502.235,Z 551.674,A -85,B 0,C 180,E1 -5845.988,E2 -5845.988} C_VEL
LIN {X 0,Y 502.182,Z 553.577,A -85,B 0,C 180,E1 -5846.792,E2 -5846.792} C_VEL
LIN {X 0,Y 502.15,Z 555.006,A -85,B 0,C 180,E1 -5847.594,E2 -5847.594} C_VEL
LIN {X 0,Y 502.067,Z 556.643,A -85,B 0,C 180,E1 -5849.199,E2 -5849.199} C_VEL
LIN {X 0,Y 502.066,Z 556.866,A -85,B 0,C 180,E1 -5850.001,E2 -5850.001} C_VEL
LIN {X 0,Y 502.066,Z 556.646,A -85,B 0,C 180,E1 -5850.803,E2 -5850.803} C_VEL
LIN {X 0,Y 502.149,Z 555.019,A -85,B 0,C 180,E1 -5852.407,E2 -5852.407} C_VEL
LIN {X 0,Y 502.182,Z 553.595,A -85,B 0,C 180,E1 -5853.21,E2 -5853.21} C_VEL
LIN {X 0,Y 502.199,Z 550.594,A -85,B 0,C 180,E1 -5854.415,E2 -5854.415} C_VEL
LIN {X 0,Y 502.281,Z 546.539,A -85,B 0,C 180,E1 -5855.621,E2 -5855.621} C_VEL
LIN {X 0,Y 502.333,Z 540.399,A -85,B 0,C 180,E1 -5857.012,E2 -5857.012} C_VEL
LIN {X 0,Y 502.495,Z 533.494,A -85,B 0,C 180,E1 -5858.243,E2 -5858.243} C_VEL
LIN {X 0,Y 502.682,Z 525.064,A -85,B 0,C 180,E1 -5859.456,E2 -5859.456} C_VEL
LIN {X 0,Y 502.95,Z 516.44,A -85,B 0,C 180,E1 -5860.467,E2 -5860.467} C_VEL
LIN {X 0,Y 503.266,Z 505.805,A -85,B 0,C 180,E1 -5861.479,E2 -5861.479} C_VEL
LIN {X 0,Y 503.588,Z 494.639,A -85,B 0,C 180,E1 -5862.336,E2 -5862.336} C_VEL
LIN {X 0,Y 503.974,Z 483.825,A -85,B 0,C 180,E1 -5862.996,E2 -5862.996} C_VEL
LIN {X 0,Y 504.31,Z 472.057,A -85,B 0,C 180,E1 -5863.551,E2 -5863.551} C_VEL
LIN {X 0,Y 504.396,Z 460.808,A -85,B 0,C 180,E1 -5863.946,E2 -5863.946} C_VEL
LIN {X 0,Y 502.926,Z 449.494,A -85,B 0,C 180,E1 -5864.259,E2 -5864.259} C_VEL
LIN {X 0,Y 502.574,Z 445.769,A -85,B 0,C 180,E1 -5864.347,E2 -5864.347} C_VEL
LIN {X 0,Y 502.792,Z 431.493,A -85,B 0,C 180,E1 -5867.49,E2 -5867.49} C_VEL
LIN {X 0,Y 502.979,Z 416.262,A -85,B 0,C 180,E1 -5870.895,E2 -5870.895} C_VEL
LIN {X 0,Y 503.252,Z 403.081,A -85,B 0,C 180,E1 -5873.891,E2 -5873.891} C_VEL
LIN {X 0,Y 503.522,Z 389.531,A -85,B 0,C 180,E1 -5877.019,E2 -5877.019} C_VEL
LIN {X 0,Y 503.815,Z 376.301,A -85,B 0,C 180,E1 -5880.145,E2 -5880.145} C_VEL
LIN {X 0,Y 504.096,Z 364.8,A -85,B 0,C 180,E1 -5882.939,E2 -5882.939} C_VEL
LIN {X 0,Y 504.517,Z 355.262,A -85,B 0,C 180,E1 -5885.318,E2 -5885.318} C_VEL
LIN {X 0,Y 504.327,Z 351.051,A -85,B 0,C 180,E1 -5886.414,E2 -5886.414} C_VEL
LIN {X 0,Y 502.814,Z 342.856,A -85,B 0,C 180,E1 -5888.697,E2 -5888.697} C_VEL
LIN {X 0,Y 502.835,Z 342.853,A -85,B 0,C 180,E1 -5892.136,E2 -5892.136} C_VEL
LIN {X 0,Y 502.805,Z 342.855,A -85,B 0,C 180,E1 -5895.469,E2 -5895.469} C_VEL
LIN {X 0,Y 502.825,Z 342.853,A -85,B 0,C 180,E1 -5898.934,E2 -5898.934} C_VEL
LIN {X 0,Y 502.799,Z 342.855,A -85,B 0,C 180,E1 -5902.046,E2 -5902.046} C_VEL
LIN {X 0,Y 502.804,Z 342.857,A -85,B 0,C 180,E1 -5905.035,E2 -5905.035} C_VEL
LIN {X 0,Y 502.793,Z 342.855,A -85,B 0,C 180,E1 -5907.916,E2 -5907.916} C_VEL
LIN {X 0,Y 502.829,Z 342.854,A -85,B 0,C 180,E1 -5910.713,E2 -5910.713} C_VEL
LIN {X 0,Y 502.868,Z 342.846,A -85,B 0,C 180,E1 -5913.44,E2 -5913.44} C_VEL
LIN {X 0,Y 502.797,Z 342.855,A -85,B 0,C 180,E1 -5916.087,E2 -5916.087} C_VEL
LIN {X 0,Y 502.789,Z 342.859,A -85,B 0,C 180,E1 -5918.689,E2 -5918.689} C_VEL
LIN {X 0,Y 502.831,Z 342.851,A -85,B 0,C 180,E1 -5921.248,E2 -5921.248} C_VEL
LIN {X 0,Y 502.854,Z 342.849,A -85,B 0,C 180,E1 -5924.601,E2 -5924.601} C_VEL
LIN {X 0,Y 502.882,Z 342.846,A -85,B 0,C 180,E1 -5928.039,E2 -5928.039} C_VEL
LIN {X 0,Y 502.876,Z 342.845,A -85,B 0,C 180,E1 -5931.157,E2 -5931.157} C_VEL
LIN {X 0,Y 502.934,Z 342.838,A -85,B 0,C 180,E1 -5933.582,E2 -5933.582} C_VEL
LIN {X 0,Y 502.901,Z 342.842,A -85,B 0,C 180,E1 -5936.796,E2 -5936.796} C_VEL
LIN {X 0,Y 503.041,Z 342.824,A -85,B 0,C 180,E1 -5939.2,E2 -5939.2} C_VEL
LIN {X 0,Y 502.909,Z 342.841,A -85,B 0,C 180,E1 -5941.602,E2 -5941.602} C_VEL
LIN {X 0,Y 502.903,Z 342.843,A -85,B 0,C 180,E1 -5943.205,E2 -5943.205} C_VEL
LIN {X 0,Y 502.934,Z 342.841,A -85,B 0,C 180,E1 -5946.419,E2 -5946.419} C_VEL
LIN {X 0,Y 502.881,Z 342.846,A -85,B 0,C 180,E1 -5948.843,E2 -5948.843} C_VEL
LIN {X 0,Y 502.853,Z 342.851,A -85,B 0,C 180,E1 -5952.102,E2 -5952.102} C_VEL
LIN {X 0,Y 502.855,Z 342.848,A -85,B 0,C 180,E1 -5955.4,E2 -5955.4} C_VEL
LIN {X 0,Y 502.853,Z 342.849,A -85,B 0,C 180,E1 -5958.122,E2 -5958.122} C_VEL
LIN {X 0,Y 502.835,Z 342.85,A -85,B 0,C 180,E1 -5960.536,E2 -5960.536} C_VEL
LIN {X 0,Y 502.801,Z 342.854,A -85,B 0,C 180,E1 -5963.04,E2 -5963.04} C_VEL
LIN {X 0,Y 502.847,Z 342.852,A -85,B 0,C 180,E1 -5965.676,E2 -5965.676} C_VEL
LIN {X 0,Y 502.844,Z 342.849,A -85,B 0,C 180,E1 -5968.373,E2 -5968.373} C_VEL
LIN {X 0,Y 502.801,Z 342.857,A -85,B 0,C 180,E1 -5971.499,E2 -5971.499} C_VEL
LIN {X 0,Y 502.811,Z 342.854,A -85,B 0,C 180,E1 -5973.994,E2 -5973.994} C_VEL
LIN {X 0,Y 502.784,Z 342.859,A -85,B 0,C 180,E1 -5977.178,E2 -5977.178} C_VEL
LIN {X 0,Y 502.795,Z 342.857,A -85,B 0,C 180,E1 -5980.015,E2 -5980.015} C_VEL
LIN {X 0,Y 502.809,Z 342.855,A -85,B 0,C 180,E1 -5982.199,E2 -5982.199} C_VEL
LIN {X 0,Y 502.808,Z 342.855,A -85,B 0,C 180,E1 -5985.468,E2 -5985.468} C_VEL
LIN {X 0,Y 502.827,Z 342.852,A -85,B 0,C 180,E1 -5988.934,E2 -5988.934} C_VEL
LIN {X 0,Y 502.797,Z 342.855,A -85,B 0,C 180,E1 -5992.046,E2 -5992.046} C_VEL
LIN {X 0,Y 502.804,Z 342.857,A -85,B 0,C 180,E1 -5995.034,E2 -5995.034} C_VEL
LIN {X 0,Y 502.815,Z 342.853,A -85,B 0,C 180,E1 -5997.223,E2 -5997.223} C_VEL
LIN {X 0,Y 502.114,Z 342.941,A -85,B 0,C 180,E1 -5997.892,E2 -5997.892} C_VEL
LIN {X 0,Y 499.249,Z 343.299,A -85,B 0,C 180,E1 -5998.978,E2 -5998.978} C_VEL
LIN {X 0,Y 496.854,Z 343.595,A -85,B 0,C 180,E1 -5999.853,E2 -5999.853} C_VEL
LIN {X 0,Y 495.837,Z 343.724,A -85,B 0,C 180,E1 -6000.528,E2 -6000.528} C_VEL
LIN {X 0,Y 495.759,Z 343.731,A -85,B 0,C 180,E1 -6000.757,E2 -6000.757} C_VEL
LIN {X 0,Y 495.798,Z 343.727,A -85,B 0,C 180,E1 -6003.932,E2 -6003.932} C_VEL
LIN {X 0,Y 495.767,Z 343.734,A -85,B 0,C 180,E1 -6007.139,E2 -6007.139} C_VEL
LIN {X 0,Y 495.778,Z 343.729,A -85,B 0,C 180,E1 -6010.109,E2 -6010.109} C_VEL
LIN {X 0,Y 495.789,Z 343.73,A -85,B 0,C 180,E1 -6012.681,E2 -6012.681} C_VEL
LIN {X 0,Y 495.797,Z 343.728,A -85,B 0,C 180,E1 -6015.217,E2 -6015.217} C_VEL
LIN {X 0,Y 495.859,Z 343.722,A -85,B 0,C 180,E1 -6018.554,E2 -6018.554} C_VEL
LIN {X 0,Y 495.88,Z 343.72,A -85,B 0,C 180,E1 -6021.852,E2 -6021.852} C_VEL
LIN {X 0,Y 495.893,Z 343.718,A -85,B 0,C 180,E1 -6023.949,E2 -6023.949} C_VEL
LIN {X 0,Y 497.851,Z 350.543,A -85,B 0,C 180,E1 -6024.278,E2 -6024.278} C_VEL
LIN {X 0,Y 497.687,Z 362.177,A -85,B 0,C 180,E1 -6024.834,E2 -6024.834} C_VEL
LIN {X 0,Y 497.387,Z 373.467,A -85,B 0,C 180,E1 -6025.542,E2 -6025.542} C_VEL
LIN {X 0,Y 497.006,Z 383.725,A -85,B 0,C 180,E1 -6026.351,E2 -6026.351} C_VEL
LIN {X 0,Y 496.649,Z 394.055,A -85,B 0,C 180,E1 -6027.363,E2 -6027.363} C_VEL
LIN {X 0,Y 496.308,Z 402.465,A -85,B 0,C 180,E1 -6028.377,E2 -6028.377} C_VEL
LIN {X 0,Y 496,Z 410.634,A -85,B 0,C 180,E1 -6029.593,E2 -6029.593} C_VEL
LIN {X 0,Y 495.714,Z 417.227,A -85,B 0,C 180,E1 -6030.812,E2 -6030.812} C_VEL
LIN {X 0,Y 495.503,Z 422.503,A -85,B 0,C 180,E1 -6032.031,E2 -6032.031} C_VEL
LIN {X 0,Y 495.406,Z 426.627,A -85,B 0,C 180,E1 -6033.252,E2 -6033.252} C_VEL
LIN {X 0,Y 495.32,Z 428.826,A -85,B 0,C 180,E1 -6034.068,E2 -6034.068} C_VEL
LIN {X 0,Y 495.282,Z 430.567,A -85,B 0,C 180,E1 -6034.883,E2 -6034.883} C_VEL
LIN {X 0,Y 495.296,Z 431.876,A -85,B 0,C 180,E1 -6035.7,E2 -6035.7} C_VEL
LIN {X 0,Y 495.26,Z 433.369,A -85,B 0,C 180,E1 -6037.337,E2 -6037.337} C_VEL
LIN {X 0,Y 495.26,Z 433.506,A -85,B 0,C 180,E1 -6038.158,E2 -6038.158} C_VEL
LIN {X 0,Y 495.214,Z 432.615,A -85,B 0,C 180,E1 -6039.805,E2 -6039.805} C_VEL
LIN {X 0,Y 495.264,Z 431.586,A -85,B 0,C 180,E1 -6040.63,E2 -6040.63} C_VEL
LIN {X 0,Y 495.378,Z 429.401,A -85,B 0,C 180,E1 -6041.785,E2 -6041.785} C_VEL
LIN {X 0,Y 495.447,Z 425.853,A -85,B 0,C 180,E1 -6043.118,E2 -6043.118} C_VEL
LIN {X 0,Y 495.597,Z 421.372,A -85,B 0,C 180,E1 -6044.368,E2 -6044.368} C_VEL
LIN {X 0,Y 495.828,Z 415.608,A -85,B 0,C 180,E1 -6045.623,E2 -6045.623} C_VEL
LIN {X 0,Y 496.062,Z 408.327,A -85,B 0,C 180,E1 -6046.883,E2 -6046.883} C_VEL
LIN {X 0,Y 496.464,Z 399.205,A -85,B 0,C 180,E1 -6048.145,E2 -6048.145} C_VEL
LIN {X 0,Y 496.778,Z 389.623,A -85,B 0,C 180,E1 -6049.203,E2 -6049.203} C_VEL
LIN {X 0,Y 497.181,Z 378.883,A -85,B 0,C 180,E1 -6050.154,E2 -6050.154} C_VEL
LIN {X 0,Y 497.561,Z 367.755,A -85,B 0,C 180,E1 -6050.938,E2 -6050.938} C_VEL
LIN {X 0,Y 497.804,Z 355.761,A -85,B 0,C 180,E1 -6051.589,E2 -6051.589} C_VEL
LIN {X 0,Y 497.846,Z 350.919,A -85,B 0,C 180,E1 -6051.804,E2 -6051.804} C_VEL
LIN {X 0,Y 495.762,Z 343.732,A -85,B 0,C 180,E1 -6052.147,E2 -6052.147} C_VEL
LIN {X 0,Y 495.791,Z 343.729,A -85,B 0,C 180,E1 -6055.166,E2 -6055.166} C_VEL
LIN {X 0,Y 495.782,Z 343.732,A -85,B 0,C 180,E1 -6057.891,E2 -6057.891} C_VEL
LIN {X 0,Y 495.754,Z 343.734,A -85,B 0,C 180,E1 -6060.686,E2 -6060.686} C_VEL
LIN {X 0,Y 495.76,Z 343.733,A -85,B 0,C 180,E1 -6063.564,E2 -6063.564} C_VEL
LIN {X 0,Y 495.729,Z 343.739,A -85,B 0,C 180,E1 -6066.543,E2 -6066.543} C_VEL
LIN {X 0,Y 495.757,Z 343.734,A -85,B 0,C 180,E1 -6069.637,E2 -6069.637} C_VEL
LIN {X 0,Y 495.741,Z 343.737,A -85,B 0,C 180,E1 -6072.507,E2 -6072.507} C_VEL
LIN {X 0,Y 495.749,Z 343.735,A -85,B 0,C 180,E1 -6075.139,E2 -6075.139} C_VEL
LIN {X 0,Y 495.76,Z 343.734,A -85,B 0,C 180,E1 -6078.219,E2 -6078.219} C_VEL
LIN {X 0,Y 495.778,Z 343.731,A -85,B 0,C 180,E1 -6081.229,E2 -6081.229} C_VEL
LIN {X 0,Y 495.757,Z 343.734,A -85,B 0,C 180,E1 -6084.463,E2 -6084.463} C_VEL
LIN {X 0,Y 495.769,Z 343.73,A -85,B 0,C 180,E1 -6087.405,E2 -6087.405} C_VEL
LIN {X 0,Y 495.78,Z 343.716,A -85,B 0,C 180,E1 -6090.254,E2 -6090.254} C_VEL
LIN {X 0,Y 495.832,Z 343.722,A -85,B 0,C 180,E1 -6093.248,E2 -6093.248} C_VEL
LIN {X 0,Y 495.751,Z 343.732,A -85,B 0,C 180,E1 -6095.725,E2 -6095.725} C_VEL
LIN {X 0,Y 495.746,Z 343.734,A -85,B 0,C 180,E1 -6098.371,E2 -6098.371} C_VEL
LIN {X 0,Y 495.783,Z 343.729,A -85,B 0,C 180,E1 -6100.971,E2 -6100.971} C_VEL
LIN {X 0,Y 495.779,Z 343.731,A -85,B 0,C 180,E1 -6103.53,E2 -6103.53} C_VEL
LIN {X 0,Y 495.797,Z 343.728,A -85,B 0,C 180,E1 -6106.055,E2 -6106.055} C_VEL
LIN {X 0,Y 495.873,Z 343.719,A -85,B 0,C 180,E1 -6108.555,E2 -6108.555} C_VEL
LIN {X 0,Y 495.871,Z 343.719,A -85,B 0,C 180,E1 -6111.852,E2 -6111.852} C_VEL
LIN {X 0,Y 495.894,Z 343.712,A -85,B 0,C 180,E1 -6114.306,E2 -6114.306} C_VEL
LIN {X 0,Y 495.991,Z 343.704,A -85,B 0,C 180,E1 -6117.563,E2 -6117.563} C_VEL
LIN {X 0,Y 495.995,Z 343.699,A -85,B 0,C 180,E1 -6120,E2 -6120} C_VEL
LIN {X 0,Y 495.991,Z 343.705,A -85,B 0,C 180,E1 -6122.436,E2 -6122.436} C_VEL
LIN {X 0,Y 495.894,Z 343.714,A -85,B 0,C 180,E1 -6125.693,E2 -6125.693} C_VEL
LIN {X 0,Y 495.87,Z 343.72,A -85,B 0,C 180,E1 -6128.148,E2 -6128.148} C_VEL
LIN {X 0,Y 495.848,Z 343.722,A -85,B 0,C 180,E1 -6131.445,E2 -6131.445} C_VEL
LIN {X 0,Y 495.787,Z 343.728,A -85,B 0,C 180,E1 -6134.783,E2 -6134.783} C_VEL
LIN {X 0,Y 495.785,Z 343.729,A -85,B 0,C 180,E1 -6137.319,E2 -6137.319} C_VEL
LIN {X 0,Y 495.775,Z 343.731,A -85,B 0,C 180,E1 -6139.89,E2 -6139.89} C_VEL
LIN {X 0,Y 495.762,Z 343.733,A -85,B 0,C 180,E1 -6142.863,E2 -6142.863} C_VEL
LIN {X 0,Y 495.797,Z 343.73,A -85,B 0,C 180,E1 -6146.067,E2 -6146.067} C_VEL
LIN {X 0,Y 495.777,Z 343.732,A -85,B 0,C 180,E1 -6148.814,E2 -6148.814} C_VEL
LIN {X 0,Y 495.757,Z 343.734,A -85,B 0,C 180,E1 -6151.727,E2 -6151.727} C_VEL
LIN {X 0,Y 495.775,Z 343.731,A -85,B 0,C 180,E1 -6154.696,E2 -6154.696} C_VEL
LIN {X 0,Y 495.733,Z 343.735,A -85,B 0,C 180,E1 -6157.561,E2 -6157.561} C_VEL
LIN {X 0,Y 495.791,Z 343.73,A -85,B 0,C 180,E1 -6160.052,E2 -6160.052} C_VEL
LIN {X 0,Y 495.762,Z 343.734,A -85,B 0,C 180,E1 -6162.879,E2 -6162.879} C_VEL
LIN {X 0,Y 495.736,Z 343.736,A -85,B 0,C 180,E1 -6166,E2 -6166} C_VEL
LIN {X 0,Y 495.771,Z 343.733,A -85,B 0,C 180,E1 -6168.705,E2 -6168.705} C_VEL
LIN {X 0,Y 495.812,Z 343.916,A -85,B 0,C 180,E1 -6170.705,E2 -6170.705} C_VEL
LIN {X 0,Y 497.701,Z 353.729,A -85,B 0,C 180,E1 -6173.625,E2 -6173.625} C_VEL
LIN {X 0,Y 497.591,Z 359.918,A -85,B 0,C 180,E1 -6175.297,E2 -6175.297} C_VEL
LIN {X 0,Y 496.964,Z 374.007,A -85,B 0,C 180,E1 -6178.924,E2 -6178.924} C_VEL
LIN {X 0,Y 496.546,Z 387.111,A -85,B 0,C 180,E1 -6182.156,E2 -6182.156} C_VEL
LIN {X 0,Y 496.276,Z 399.017,A -85,B 0,C 180,E1 -6185.004,E2 -6185.004} C_VEL
LIN {X 0,Y 496.011,Z 411.631,A -85,B 0,C 180,E1 -6187.947,E2 -6187.947} C_VEL
LIN {X 0,Y 495.76,Z 424.861,A -85,B 0,C 180,E1 -6190.971,E2 -6190.971} C_VEL
LIN {X 0,Y 495.573,Z 436.202,A -85,B 0,C 180,E1 -6193.524,E2 -6193.524} C_VEL
LIN {X 0,Y 495.498,Z 444.753,A -85,B 0,C 180,E1 -6195.445,E2 -6195.445} C_VEL
LIN {X 0,Y 496.951,Z 458.405,A -85,B 0,C 180,E1 -6195.802,E2 -6195.802} C_VEL
LIN {X 0,Y 497.541,Z 463.48,A -85,B 0,C 180,E1 -6195.976,E2 -6195.976} C_VEL
LIN {X 0,Y 497.202,Z 476.868,A -85,B 0,C 180,E1 -6196.513,E2 -6196.513} C_VEL
LIN {X 0,Y 496.841,Z 488.054,A -85,B 0,C 180,E1 -6197.123,E2 -6197.123} C_VEL
LIN {X 0,Y 496.491,Z 499.872,A -85,B 0,C 180,E1 -6197.949,E2 -6197.949} C_VEL
LIN {X 0,Y 496.076,Z 510.453,A -85,B 0,C 180,E1 -6198.871,E2 -6198.871} C_VEL
LIN {X 0,Y 495.778,Z 519.128,A -85,B 0,C 180,E1 -6199.794,E2 -6199.794} C_VEL
LIN {X 0,Y 495.528,Z 527.149,A -85,B 0,C 180,E1 -6200.819,E2 -6200.819} C_VEL
LIN {X 0,Y 495.357,Z 535.006,A -85,B 0,C 180,E1 -6202.049,E2 -6202.049} C_VEL
LIN {X 0,Y 495.203,Z 542.254,A -85,B 0,C 180,E1 -6203.481,E2 -6203.481} C_VEL
LIN {X 0,Y 495.138,Z 547.088,A -85,B 0,C 180,E1 -6204.707,E2 -6204.707} C_VEL
LIN {X 0,Y 495.169,Z 550.794,A -85,B 0,C 180,E1 -6205.931,E2 -6205.931} C_VEL
LIN {X 0,Y 495.134,Z 552.7,A -85,B 0,C 180,E1 -6206.746,E2 -6206.746} C_VEL
LIN {X 0,Y 495.095,Z 554.13,A -85,B 0,C 180,E1 -6207.56,E2 -6207.56} C_VEL
LIN {X 0,Y 495.019,Z 555.77,A -85,B 0,C 180,E1 -6209.187,E2 -6209.187} C_VEL
LIN {X 0,Y 495.02,Z 555.995,A -85,B 0,C 180,E1 -6210.001,E2 -6210.001} C_VEL
LIN {X 0,Y 495.019,Z 555.775,A -85,B 0,C 180,E1 -6210.814,E2 -6210.814} C_VEL
LIN {X 0,Y 495.094,Z 554.149,A -85,B 0,C 180,E1 -6212.441,E2 -6212.441} C_VEL
LIN {X 0,Y 495.134,Z 552.725,A -85,B 0,C 180,E1 -6213.255,E2 -6213.255} C_VEL
LIN {X 0,Y 495.133,Z 549.722,A -85,B 0,C 180,E1 -6214.478,E2 -6214.478} C_VEL
LIN {X 0,Y 495.21,Z 544.485,A -85,B 0,C 180,E1 -6215.999,E2 -6215.999} C_VEL
LIN {X 0,Y 495.274,Z 538.388,A -85,B 0,C 180,E1 -6217.338,E2 -6217.338} C_VEL
LIN {X 0,Y 495.455,Z 531.359,A -85,B 0,C 180,E1 -6218.566,E2 -6218.566} C_VEL
LIN {X 0,Y 495.659,Z 522.568,A -85,B 0,C 180,E1 -6219.797,E2 -6219.797} C_VEL
LIN {X 0,Y 495.985,Z 513.585,A -85,B 0,C 180,E1 -6220.822,E2 -6220.822} C_VEL
LIN {X 0,Y 496.375,Z 502.55,A -85,B 0,C 180,E1 -6221.848,E2 -6221.848} C_VEL
LIN {X 0,Y 496.692,Z 492.065,A -85,B 0,C 180,E1 -6222.628,E2 -6222.628} C_VEL
LIN {X 0,Y 497.069,Z 479.996,A -85,B 0,C 180,E1 -6223.335,E2 -6223.335} C_VEL
LIN {X 0,Y 497.456,Z 467.254,A -85,B 0,C 180,E1 -6223.897,E2 -6223.897} C_VEL
LIN {X 0,Y 497.413,Z 461.239,A -85,B 0,C 180,E1 -6224.107,E2 -6224.107} C_VEL
LIN {X 0,Y 496.052,Z 450.564,A -85,B 0,C 180,E1 -6224.422,E2 -6224.422} C_VEL
LIN {X 0,Y 495.505,Z 444.878,A -85,B 0,C 180,E1 -6224.556,E2 -6224.556} C_VEL
LIN {X 0,Y 495.702,Z 430.675,A -85,B 0,C 180,E1 -6227.748,E2 -6227.748} C_VEL
LIN {X 0,Y 495.922,Z 417.507,A -85,B 0,C 180,E1 -6230.751,E2 -6230.751} C_VEL
LIN {X 0,Y 496.178,Z 404.227,A -85,B 0,C 180,E1 -6233.809,E2 -6233.809} C_VEL
LIN {X 0,Y 496.453,Z 390.867,A -85,B 0,C 180,E1 -6236.937,E2 -6236.937} C_VEL
LIN {X 0,Y 496.795,Z 378.011,A -85,B 0,C 180,E1 -6240.018,E2 -6240.018} C_VEL
LIN {X 0,Y 497.126,Z 365.999,A -85,B 0,C 180,E1 -6242.976,E2 -6242.976} C_VEL
LIN {X 0,Y 497.58,Z 354.636,A -85,B 0,C 180,E1 -6245.865,E2 -6245.865} C_VEL
LIN {X 0,Y 496.652,Z 348.349,A -85,B 0,C 180,E1 -6247.586,E2 -6247.586} C_VEL
LIN {X 0,Y 495.792,Z 343.73,A -85,B 0,C 180,E1 -6248.933,E2 -6248.933} C_VEL
LIN {X 0,Y 495.782,Z 343.732,A -85,B 0,C 180,E1 -6251.779,E2 -6251.779} C_VEL
LIN {X 0,Y 495.754,Z 343.735,A -85,B 0,C 180,E1 -6255.14,E2 -6255.14} C_VEL
LIN {X 0,Y 495.761,Z 343.732,A -85,B 0,C 180,E1 -6258.219,E2 -6258.219} C_VEL
LIN {X 0,Y 495.756,Z 343.734,A -85,B 0,C 180,E1 -6261.409,E2 -6261.409} C_VEL
LIN {X 0,Y 495.753,Z 343.734,A -85,B 0,C 180,E1 -6264.463,E2 -6264.463} C_VEL
LIN {X 0,Y 495.775,Z 343.731,A -85,B 0,C 180,E1 -6267.406,E2 -6267.406} C_VEL
LIN {X 0,Y 495.771,Z 343.731,A -85,B 0,C 180,E1 -6270.254,E2 -6270.254} C_VEL
LIN {X 0,Y 495.829,Z 343.723,A -85,B 0,C 180,E1 -6273.251,E2 -6273.251} C_VEL
LIN {X 0,Y 495.758,Z 343.731,A -85,B 0,C 180,E1 -6275.725,E2 -6275.725} C_VEL
LIN {X 0,Y 495.753,Z 343.734,A -85,B 0,C 180,E1 -6278.372,E2 -6278.372} C_VEL
LIN {X 0,Y 495.787,Z 343.729,A -85,B 0,C 180,E1 -6280.972,E2 -6280.972} C_VEL
LIN {X 0,Y 495.813,Z 343.728,A -85,B 0,C 180,E1 -6284.376,E2 -6284.376} C_VEL
LIN {X 0,Y 495.789,Z 343.729,A -85,B 0,C 180,E1 -6286.891,E2 -6286.891} C_VEL
LIN {X 0,Y 495.779,Z 343.729,A -85,B 0,C 180,E1 -6289.381,E2 -6289.381} C_VEL
LIN {X 0,Y 495.878,Z 343.717,A -85,B 0,C 180,E1 -6291.852,E2 -6291.852} C_VEL
LIN {X 0,Y 495.902,Z 343.717,A -85,B 0,C 180,E1 -6294.307,E2 -6294.307} C_VEL
LIN {X 0,Y 495.997,Z 343.703,A -85,B 0,C 180,E1 -6297.564,E2 -6297.564} C_VEL
LIN {X 0,Y 496.005,Z 343.704,A -85,B 0,C 180,E1 -6300,E2 -6300} C_VEL
LIN {X 0,Y 495.999,Z 343.703,A -85,B 0,C 180,E1 -6302.436,E2 -6302.436} C_VEL
LIN {X 0,Y 495.9,Z 343.717,A -85,B 0,C 180,E1 -6305.694,E2 -6305.694} C_VEL
LIN {X 0,Y 495.88,Z 343.718,A -85,B 0,C 180,E1 -6308.148,E2 -6308.148} C_VEL
LIN {X 0,Y 495.858,Z 343.721,A -85,B 0,C 180,E1 -6311.445,E2 -6311.445} C_VEL
LIN {X 0,Y 495.797,Z 343.727,A -85,B 0,C 180,E1 -6314.783,E2 -6314.783} C_VEL
LIN {X 0,Y 495.793,Z 343.728,A -85,B 0,C 180,E1 -6317.319,E2 -6317.319} C_VEL
LIN {X 0,Y 495.778,Z 343.732,A -85,B 0,C 180,E1 -6319.89,E2 -6319.89} C_VEL
LIN {X 0,Y 495.768,Z 343.73,A -85,B 0,C 180,E1 -6322.861,E2 -6322.861} C_VEL
LIN {X 0,Y 495.798,Z 343.728,A -85,B 0,C 180,E1 -6326.068,E2 -6326.068} C_VEL
LIN {X 0,Y 495.776,Z 343.729,A -85,B 0,C 180,E1 -6328.815,E2 -6328.815} C_VEL
LIN {X 0,Y 495.763,Z 343.733,A -85,B 0,C 180,E1 -6331.725,E2 -6331.725} C_VEL
LIN {X 0,Y 495.776,Z 343.73,A -85,B 0,C 180,E1 -6334.694,E2 -6334.694} C_VEL
LIN {X 0,Y 495.736,Z 343.736,A -85,B 0,C 180,E1 -6337.562,E2 -6337.562} C_VEL
LIN {X 0,Y 495.773,Z 343.73,A -85,B 0,C 180,E1 -6340.7,E2 -6340.7} C_VEL
LIN {X 0,Y 495.74,Z 343.734,A -85,B 0,C 180,E1 -6344.001,E2 -6344.001} C_VEL
LIN {X 0,Y 495.733,Z 343.738,A -85,B 0,C 180,E1 -6347.117,E2 -6347.117} C_VEL
LIN {X 0,Y 495.765,Z 343.732,A -85,B 0,C 180,E1 -6349.953,E2 -6349.953} C_VEL
LIN {X 0,Y 495.725,Z 343.737,A -85,B 0,C 180,E1 -6352.554,E2 -6352.554} C_VEL
LIN {X 0,Y 495.784,Z 343.73,A -85,B 0,C 180,E1 -6355.457,E2 -6355.457} C_VEL
LIN {X 0,Y 495.763,Z 343.733,A -85,B 0,C 180,E1 -6358.364,E2 -6358.364} C_VEL
LIN {X 0,Y 495.759,Z 343.731,A -85,B 0,C 180,E1 -6360.757,E2 -6360.757} C_VEL
LIN {X 0,Y 495.102,Z 343.816,A -85,B 0,C 180,E1 -6361.436,E2 -6361.436} C_VEL
LIN {X 0,Y 492.246,Z 344.17,A -85,B 0,C 180,E1 -6362.539,E2 -6362.539} C_VEL
LIN {X 0,Y 489.838,Z 344.471,A -85,B 0,C 180,E1 -6363.427,E2 -6363.427} C_VEL
LIN {X 0,Y 488.822,Z 344.596,A -85,B 0,C 180,E1 -6364.114,E2 -6364.114} C_VEL
LIN {X 0,Y 488.749,Z 344.605,A -85,B 0,C 180,E1 -6364.346,E2 -6364.346} C_VEL
LIN {X 0,Y 488.73,Z 344.61,A -85,B 0,C 180,E1 -6367.153,E2 -6367.153} C_VEL
LIN {X 0,Y 488.732,Z 344.606,A -85,B 0,C 180,E1 -6369.81,E2 -6369.81} C_VEL
LIN {X 0,Y 488.737,Z 344.607,A -85,B 0,C 180,E1 -6372.423,E2 -6372.423} C_VEL
LIN {X 0,Y 488.769,Z 344.605,A -85,B 0,C 180,E1 -6374.999,E2 -6374.999} C_VEL
LIN {X 0,Y 488.813,Z 344.599,A -85,B 0,C 180,E1 -6378.387,E2 -6378.387} C_VEL
LIN {X 0,Y 488.824,Z 344.598,A -85,B 0,C 180,E1 -6381.733,E2 -6381.733} C_VEL
LIN {X 0,Y 488.868,Z 344.777,A -85,B 0,C 180,E1 -6383.758,E2 -6383.758} C_VEL
LIN {X 0,Y 491.048,Z 352.893,A -85,B 0,C 180,E1 -6384.147,E2 -6384.147} C_VEL
LIN {X 0,Y 490.78,Z 364.988,A -85,B 0,C 180,E1 -6384.762,E2 -6384.762} C_VEL
LIN {X 0,Y 490.407,Z 377.26,A -85,B 0,C 180,E1 -6385.582,E2 -6385.582} C_VEL
LIN {X 0,Y 489.991,Z 388.065,A -85,B 0,C 180,E1 -6386.505,E2 -6386.505} C_VEL
LIN {X 0,Y 489.6,Z 397.698,A -85,B 0,C 180,E1 -6387.531,E2 -6387.531} C_VEL
LIN {X 0,Y 489.202,Z 407.047,A -85,B 0,C 180,E1 -6388.765,E2 -6388.765} C_VEL
LIN {X 0,Y 488.892,Z 414.495,A -85,B 0,C 180,E1 -6389.999,E2 -6389.999} C_VEL
LIN {X 0,Y 488.591,Z 420.499,A -85,B 0,C 180,E1 -6391.236,E2 -6391.236} C_VEL
LIN {X 0,Y 488.468,Z 425.255,A -85,B 0,C 180,E1 -6392.473,E2 -6392.473} C_VEL
LIN {X 0,Y 488.363,Z 428.935,A -85,B 0,C 180,E1 -6393.712,E2 -6393.712} C_VEL
LIN {X 0,Y 488.243,Z 431.634,A -85,B 0,C 180,E1 -6394.954,E2 -6394.954} C_VEL
LIN {X 0,Y 488.26,Z 432.899,A -85,B 0,C 180,E1 -6395.782,E2 -6395.782} C_VEL
LIN {X 0,Y 488.225,Z 433.832,A -85,B 0,C 180,E1 -6396.654,E2 -6396.654} C_VEL
LIN {X 0,Y 488.239,Z 434.278,A -85,B 0,C 180,E1 -6397.443,E2 -6397.443} C_VEL
LIN {X 0,Y 488.193,Z 434.058,A -85,B 0,C 180,E1 -6399.111,E2 -6399.111} C_VEL
LIN {X 0,Y 488.177,Z 433.379,A -85,B 0,C 180,E1 -6399.948,E2 -6399.948} C_VEL
LIN {X 0,Y 488.254,Z 432.269,A -85,B 0,C 180,E1 -6400.784,E2 -6400.784} C_VEL
LIN {X 0,Y 488.368,Z 430.188,A -85,B 0,C 180,E1 -6401.879,E2 -6401.879} C_VEL
LIN {X 0,Y 488.443,Z 426.362,A -85,B 0,C 180,E1 -6403.309,E2 -6403.309} C_VEL
LIN {X 0,Y 488.636,Z 421.755,A -85,B 0,C 180,E1 -6404.578,E2 -6404.578} C_VEL
LIN {X 0,Y 488.919,Z 414.74,A -85,B 0,C 180,E1 -6406.063,E2 -6406.063} C_VEL
LIN {X 0,Y 489.244,Z 407.056,A -85,B 0,C 180,E1 -6407.341,E2 -6407.341} C_VEL
LIN {X 0,Y 489.648,Z 397.987,A -85,B 0,C 180,E1 -6408.54,E2 -6408.54} C_VEL
LIN {X 0,Y 489.974,Z 388.21,A -85,B 0,C 180,E1 -6409.589,E2 -6409.589} C_VEL
LIN {X 0,Y 490.335,Z 378.286,A -85,B 0,C 180,E1 -6410.448,E2 -6410.448} C_VEL
LIN {X 0,Y 490.719,Z 367.436,A -85,B 0,C 180,E1 -6411.196,E2 -6411.196} C_VEL
LIN {X 0,Y 491.015,Z 355.254,A -85,B 0,C 180,E1 -6411.847,E2 -6411.847} C_VEL
LIN {X 0,Y 491.075,Z 352.893,A -85,B 0,C 180,E1 -6411.955,E2 -6411.955} C_VEL
LIN {X 0,Y 488.713,Z 344.61,A -85,B 0,C 180,E1 -6412.362,E2 -6412.362} C_VEL
LIN {X 0,Y 488.75,Z 344.608,A -85,B 0,C 180,E1 -6415.555,E2 -6415.555} C_VEL
LIN {X 0,Y 488.746,Z 344.609,A -85,B 0,C 180,E1 -6418.328,E2 -6418.328} C_VEL
LIN {X 0,Y 488.694,Z 344.613,A -85,B 0,C 180,E1 -6421.179,E2 -6421.179} C_VEL
LIN {X 0,Y 488.732,Z 344.607,A -85,B 0,C 180,E1 -6424.112,E2 -6424.112} C_VEL
LIN {X 0,Y 488.68,Z 344.616,A -85,B 0,C 180,E1 -6427.158,E2 -6427.158} C_VEL
LIN {X 0,Y 488.718,Z 344.61,A -85,B 0,C 180,E1 -6430.344,E2 -6430.344} C_VEL
LIN {X 0,Y 488.716,Z 344.611,A -85,B 0,C 180,E1 -6432.826,E2 -6432.826} C_VEL
LIN {X 0,Y 488.699,Z 344.613,A -85,B 0,C 180,E1 -6435.975,E2 -6435.975} C_VEL
LIN {X 0,Y 488.713,Z 344.613,A -85,B 0,C 180,E1 -6438.584,E2 -6438.584} C_VEL
LIN {X 0,Y 488.747,Z 344.607,A -85,B 0,C 180,E1 -6440.94,E2 -6440.94} C_VEL
LIN {X 0,Y 488.685,Z 344.612,A -85,B 0,C 180,E1 -6443.868,E2 -6443.868} C_VEL
LIN {X 0,Y 488.738,Z 344.606,A -85,B 0,C 180,E1 -6446.877,E2 -6446.877} C_VEL
LIN {X 0,Y 488.733,Z 344.593,A -85,B 0,C 180,E1 -6449.781,E2 -6449.781} C_VEL
LIN {X 0,Y 488.797,Z 344.598,A -85,B 0,C 180,E1 -6453.054,E2 -6453.054} C_VEL
LIN {X 0,Y 488.692,Z 344.612,A -85,B 0,C 180,E1 -6456.254,E2 -6456.254} C_VEL
LIN {X 0,Y 488.744,Z 344.607,A -85,B 0,C 180,E1 -6459.175,E2 -6459.175} C_VEL
LIN {X 0,Y 488.756,Z 344.602,A -85,B 0,C 180,E1 -6461.627,E2 -6461.627} C_VEL
LIN {X 0,Y 488.762,Z 344.605,A -85,B 0,C 180,E1 -6464.999,E2 -6464.999} C_VEL
LIN {X 0,Y 488.833,Z 344.597,A -85,B 0,C 180,E1 -6468.388,E2 -6468.388} C_VEL
LIN {X 0,Y 488.816,Z 344.598,A -85,B 0,C 180,E1 -6471.733,E2 -6471.733} C_VEL
LIN {X 0,Y 488.853,Z 344.589,A -85,B 0,C 180,E1 -6474.224,E2 -6474.224} C_VEL
LIN {X 0,Y 488.959,Z 344.58,A -85,B 0,C 180,E1 -6477.528,E2 -6477.528} C_VEL
LIN {X 0,Y 488.967,Z 344.575,A -85,B 0,C 180,E1 -6480,E2 -6480} C_VEL
LIN {X 0,Y 488.959,Z 344.581,A -85,B 0,C 180,E1 -6482.471,E2 -6482.471} C_VEL
LIN {X 0,Y 488.853,Z 344.591,A -85,B 0,C 180,E1 -6485.776,E2 -6485.776} C_VEL
LIN {X 0,Y 488.814,Z 344.599,A -85,B 0,C 180,E1 -6488.266,E2 -6488.266} C_VEL
LIN {X 0,Y 488.802,Z 344.599,A -85,B 0,C 180,E1 -6491.612,E2 -6491.612} C_VEL
LIN {X 0,Y 488.758,Z 344.604,A -85,B 0,C 180,E1 -6495,E2 -6495} C_VEL
LIN {X 0,Y 488.751,Z 344.606,A -85,B 0,C 180,E1 -6498.442,E2 -6498.442} C_VEL
LIN {X 0,Y 488.703,Z 344.611,A -85,B 0,C 180,E1 -6501.071,E2 -6501.071} C_VEL
LIN {X 0,Y 488.69,Z 344.612,A -85,B 0,C 180,E1 -6503.746,E2 -6503.746} C_VEL
LIN {X 0,Y 488.796,Z 344.602,A -85,B 0,C 180,E1 -6506.946,E2 -6506.946} C_VEL
LIN {X 0,Y 488.716,Z 344.612,A -85,B 0,C 180,E1 -6510.365,E2 -6510.365} C_VEL
LIN {X 0,Y 488.733,Z 344.609,A -85,B 0,C 180,E1 -6513.485,E2 -6513.485} C_VEL
LIN {X 0,Y 488.688,Z 344.615,A -85,B 0,C 180,E1 -6516.356,E2 -6516.356} C_VEL
LIN {X 0,Y 488.747,Z 344.605,A -85,B 0,C 180,E1 -6519.25,E2 -6519.25} C_VEL
LIN {X 0,Y 488.733,Z 344.609,A -85,B 0,C 180,E1 -6522.521,E2 -6522.521} C_VEL
LIN {X 0,Y 488.701,Z 344.612,A -85,B 0,C 180,E1 -6525.976,E2 -6525.976} C_VEL
LIN {X 0,Y 488.726,Z 344.611,A -85,B 0,C 180,E1 -6528.587,E2 -6528.587} C_VEL
LIN {X 0,Y 488.771,Z 344.712,A -85,B 0,C 180,E1 -6530.387,E2 -6530.387} C_VEL
LIN {X 0,Y 490.622,Z 354.431,A -85,B 0,C 180,E1 -6533.339,E2 -6533.339} C_VEL
LIN {X 0,Y 490.783,Z 358.324,A -85,B 0,C 180,E1 -6534.434,E2 -6534.434} C_VEL
LIN {X 0,Y 490.169,Z 369.619,A -85,B 0,C 180,E1 -6537.436,E2 -6537.436} C_VEL
LIN {X 0,Y 489.761,Z 380.904,A -85,B 0,C 180,E1 -6540.326,E2 -6540.326} C_VEL
LIN {X 0,Y 489.358,Z 394,A -85,B 0,C 180,E1 -6543.564,E2 -6543.564} C_VEL
LIN {X 0,Y 489.053,Z 406.759,A -85,B 0,C 180,E1 -6546.63,E2 -6546.63} C_VEL
LIN {X 0,Y 488.794,Z 420.318,A -85,B 0,C 180,E1 -6549.814,E2 -6549.814} C_VEL
LIN {X 0,Y 488.581,Z 433.468,A -85,B 0,C 180,E1 -6552.85,E2 -6552.85} C_VEL
LIN {X 0,Y 488.423,Z 443.882,A -85,B 0,C 180,E1 -6555.23,E2 -6555.23} C_VEL
LIN {X 0,Y 490.029,Z 459.347,A -85,B 0,C 180,E1 -6555.65,E2 -6555.65} C_VEL
LIN {X 0,Y 490.562,Z 464.879,A -85,B 0,C 180,E1 -6555.852,E2 -6555.852} C_VEL
LIN {X 0,Y 490.138,Z 478,A -85,B 0,C 180,E1 -6556.421,E2 -6556.421} C_VEL
LIN {X 0,Y 489.77,Z 489.309,A -85,B 0,C 180,E1 -6557.076,E2 -6557.076} C_VEL
LIN {X 0,Y 489.454,Z 500.283,A -85,B 0,C 180,E1 -6557.878,E2 -6557.878} C_VEL
LIN {X 0,Y 489.012,Z 510.618,A -85,B 0,C 180,E1 -6558.813,E2 -6558.813} C_VEL
LIN {X 0,Y 488.694,Z 519.945,A -85,B 0,C 180,E1 -6559.854,E2 -6559.854} C_VEL
LIN {X 0,Y 488.397,Z 529.048,A -85,B 0,C 180,E1 -6561.102,E2 -6561.102} C_VEL
LIN {X 0,Y 488.24,Z 536.4,A -85,B 0,C 180,E1 -6562.349,E2 -6562.349} C_VEL
LIN {X 0,Y 488.125,Z 542.783,A -85,B 0,C 180,E1 -6563.72,E2 -6563.72} C_VEL
LIN {X 0,Y 488.025,Z 547.546,A -85,B 0,C 180,E1 -6565.044,E2 -6565.044} C_VEL
LIN {X 0,Y 488.106,Z 549.914,A -85,B 0,C 180,E1 -6565.872,E2 -6565.872} C_VEL
LIN {X 0,Y 488.086,Z 551.824,A -85,B 0,C 180,E1 -6566.699,E2 -6566.699} C_VEL
LIN {X 0,Y 488.041,Z 553.254,A -85,B 0,C 180,E1 -6567.525,E2 -6567.525} C_VEL
LIN {X 0,Y 487.995,Z 554.274,A -85,B 0,C 180,E1 -6568.35,E2 -6568.35} C_VEL
LIN {X 0,Y 487.972,Z 554.898,A -85,B 0,C 180,E1 -6569.175,E2 -6569.175} C_VEL
LIN {X 0,Y 487.974,Z 555.123,A -85,B 0,C 180,E1 -6570.001,E2 -6570.001} C_VEL
LIN {X 0,Y 487.971,Z 554.905,A -85,B 0,C 180,E1 -6570.826,E2 -6570.826} C_VEL
LIN {X 0,Y 487.994,Z 554.289,A -85,B 0,C 180,E1 -6571.651,E2 -6571.651} C_VEL
LIN {X 0,Y 488.039,Z 553.278,A -85,B 0,C 180,E1 -6572.477,E2 -6572.477} C_VEL
LIN {X 0,Y 488.085,Z 551.855,A -85,B 0,C 180,E1 -6573.302,E2 -6573.302} C_VEL
LIN {X 0,Y 488.07,Z 548.85,A -85,B 0,C 180,E1 -6574.543,E2 -6574.543} C_VEL
LIN {X 0,Y 488.154,Z 544.794,A -85,B 0,C 180,E1 -6575.785,E2 -6575.785} C_VEL
LIN {X 0,Y 488.182,Z 538.544,A -85,B 0,C 180,E1 -6577.237,E2 -6577.237} C_VEL
LIN {X 0,Y 488.358,Z 531.741,A -85,B 0,C 180,E1 -6578.483,E2 -6578.483} C_VEL
LIN {X 0,Y 488.566,Z 523.308,A -85,B 0,C 180,E1 -6579.732,E2 -6579.732} C_VEL
LIN {X 0,Y 488.872,Z 514.684,A -85,B 0,C 180,E1 -6580.772,E2 -6580.772} C_VEL
LIN {X 0,Y 489.275,Z 504.068,A -85,B 0,C 180,E1 -6581.811,E2 -6581.811} C_VEL
LIN {X 0,Y 489.662,Z 492.546,A -85,B 0,C 180,E1 -6582.717,E2 -6582.717} C_VEL
LIN {X 0,Y 490.077,Z 480.121,A -85,B 0,C 180,E1 -6583.476,E2 -6583.476} C_VEL
LIN {X 0,Y 490.494,Z 467.688,A -85,B 0,C 180,E1 -6584.046,E2 -6584.046} C_VEL
LIN {X 0,Y 490.422,Z 461.895,A -85,B 0,C 180,E1 -6584.26,E2 -6584.26} C_VEL
LIN {X 0,Y 489.127,Z 450.832,A -85,B 0,C 180,E1 -6584.604,E2 -6584.604} C_VEL
LIN {X 0,Y 488.428,Z 444.012,A -85,B 0,C 180,E1 -6584.772,E2 -6584.772} C_VEL
LIN {X 0,Y 488.624,Z 430.152,A -85,B 0,C 180,E1 -6587.954,E2 -6587.954} C_VEL
LIN {X 0,Y 488.854,Z 416.722,A -85,B 0,C 180,E1 -6591.065,E2 -6591.065} C_VEL
LIN {X 0,Y 489.145,Z 403.452,A -85,B 0,C 180,E1 -6594.173,E2 -6594.173} C_VEL
LIN {X 0,Y 489.492,Z 390.107,A -85,B 0,C 180,E1 -6597.352,E2 -6597.352} C_VEL
LIN {X 0,Y 489.843,Z 376.861,A -85,B 0,C 180,E1 -6600.588,E2 -6600.588} C_VEL
LIN {X 0,Y 490.163,Z 365.744,A -85,B 0,C 180,E1 -6603.382,E2 -6603.382} C_VEL
LIN {X 0,Y 490.611,Z 355.742,A -85,B 0,C 180,E1 -6605.968,E2 -6605.968} C_VEL
LIN {X 0,Y 489.574,Z 348.998,A -85,B 0,C 180,E1 -6607.857,E2 -6607.857} C_VEL
LIN {X 0,Y 488.75,Z 344.608,A -85,B 0,C 180,E1 -6609.152,E2 -6609.152} C_VEL
LIN {X 0,Y 488.7,Z 344.615,A -85,B 0,C 180,E1 -6612.525,E2 -6612.525} C_VEL
LIN {X 0,Y 488.717,Z 344.611,A -85,B 0,C 180,E1 -6615.199,E2 -6615.199} C_VEL
LIN {X 0,Y 488.712,Z 344.61,A -85,B 0,C 180,E1 -6618.4,E2 -6618.4} C_VEL
LIN {X 0,Y 488.71,Z 344.612,A -85,B 0,C 180,E1 -6620.947,E2 -6620.947} C_VEL
LIN {X 0,Y 488.682,Z 344.614,A -85,B 0,C 180,E1 -6623.868,E2 -6623.868} C_VEL
LIN {X 0,Y 488.744,Z 344.607,A -85,B 0,C 180,E1 -6626.878,E2 -6626.878} C_VEL
LIN {X 0,Y 488.729,Z 344.608,A -85,B 0,C 180,E1 -6629.781,E2 -6629.781} C_VEL
LIN {X 0,Y 488.797,Z 344.601,A -85,B 0,C 180,E1 -6633.057,E2 -6633.057} C_VEL
LIN {X 0,Y 488.699,Z 344.612,A -85,B 0,C 180,E1 -6636.255,E2 -6636.255} C_VEL
LIN {X 0,Y 488.752,Z 344.605,A -85,B 0,C 180,E1 -6639.176,E2 -6639.176} C_VEL
LIN {X 0,Y 488.754,Z 344.604,A -85,B 0,C 180,E1 -6641.632,E2 -6641.632} C_VEL
LIN {X 0,Y 488.768,Z 344.604,A -85,B 0,C 180,E1 -6645,E2 -6645} C_VEL
LIN {X 0,Y 488.811,Z 344.599,A -85,B 0,C 180,E1 -6648.388,E2 -6648.388} C_VEL
LIN {X 0,Y 488.822,Z 344.595,A -85,B 0,C 180,E1 -6651.734,E2 -6651.734} C_VEL
LIN {X 0,Y 488.861,Z 344.594,A -85,B 0,C 180,E1 -6654.224,E2 -6654.224} C_VEL
LIN {X 0,Y 488.965,Z 344.578,A -85,B 0,C 180,E1 -6657.529,E2 -6657.529} C_VEL
LIN {X 0,Y 488.961,Z 344.58,A -85,B 0,C 180,E1 -6660.824,E2 -6660.824} C_VEL
LIN {X 0,Y 488.967,Z 344.579,A -85,B 0,C 180,E1 -6662.472,E2 -6662.472} C_VEL
LIN {X 0,Y 488.86,Z 344.593,A -85,B 0,C 180,E1 -6665.776,E2 -6665.776} C_VEL
LIN {X 0,Y 488.824,Z 344.597,A -85,B 0,C 180,E1 -6668.266,E2 -6668.266} C_VEL
LIN {X 0,Y 488.812,Z 344.598,A -85,B 0,C 180,E1 -6671.613,E2 -6671.613} C_VEL
LIN {X 0,Y 488.769,Z 344.602,A -85,B 0,C 180,E1 -6675,E2 -6675} C_VEL
LIN {X 0,Y 488.762,Z 344.604,A -85,B 0,C 180,E1 -6678.442,E2 -6678.442} C_VEL
LIN {X 0,Y 488.713,Z 344.609,A -85,B 0,C 180,E1 -6681.071,E2 -6681.071} C_VEL
LIN {X 0,Y 488.7,Z 344.613,A -85,B 0,C 180,E1 -6683.745,E2 -6683.745} C_VEL
LIN {X 0,Y 488.798,Z 344.6,A -85,B 0,C 180,E1 -6686.944,E2 -6686.944} C_VEL
LIN {X 0,Y 488.716,Z 344.609,A -85,B 0,C 180,E1 -6690.363,E2 -6690.363} C_VEL
LIN {X 0,Y 488.741,Z 344.609,A -85,B 0,C 180,E1 -6693.484,E2 -6693.484} C_VEL
LIN {X 0,Y 488.689,Z 344.612,A -85,B 0,C 180,E1 -6696.354,E2 -6696.354} C_VEL
LIN {X 0,Y 488.709,Z 344.613,A -85,B 0,C 180,E1 -6699.254,E2 -6699.254} C_VEL
LIN {X 0,Y 488.714,Z 344.611,A -85,B 0,C 180,E1 -6701.6,E2 -6701.6} C_VEL
LIN {X 0,Y 488.719,Z 344.61,A -85,B 0,C 180,E1 -6704.801,E2 -6704.801} C_VEL
LIN {X 0,Y 488.699,Z 344.612,A -85,B 0,C 180,E1 -6707.474,E2 -6707.474} C_VEL
LIN {X 0,Y 488.74,Z 344.607,A -85,B 0,C 180,E1 -6709.676,E2 -6709.676} C_VEL
LIN {X 0,Y 488.677,Z 344.616,A -85,B 0,C 180,E1 -6712.84,E2 -6712.84} C_VEL
LIN {X 0,Y 488.737,Z 344.607,A -85,B 0,C 180,E1 -6715.887,E2 -6715.887} C_VEL
LIN {X 0,Y 488.699,Z 344.612,A -85,B 0,C 180,E1 -6718.82,E2 -6718.82} C_VEL
LIN {X 0,Y 488.751,Z 344.605,A -85,B 0,C 180,E1 -6721.671,E2 -6721.671} C_VEL
LIN {X 0,Y 488.749,Z 344.605,A -85,B 0,C 180,E1 -6724.346,E2 -6724.346} C_VEL
LIN {X 0,Y 488.105,Z 344.688,A -85,B 0,C 180,E1 -6725.034,E2 -6725.034} C_VEL
LIN {X 0,Y 485.236,Z 345.045,A -85,B 0,C 180,E1 -6726.15,E2 -6726.15} C_VEL
LIN {X 0,Y 482.789,Z 345.35,A -85,B 0,C 180,E1 -6727.05,E2 -6727.05} C_VEL
LIN {X 0,Y 481.731,Z 345.478,A -85,B 0,C 180,E1 -6727.745,E2 -6727.745} C_VEL
LIN {X 0,Y 481.642,Z 345.489,A -85,B 0,C 180,E1 -6727.981,E2 -6727.981} C_VEL
LIN {X 0,Y 481.712,Z 345.482,A -85,B 0,C 180,E1 -6730.393,E2 -6730.393} C_VEL
LIN {X 0,Y 481.696,Z 345.485,A -85,B 0,C 180,E1 -6733.033,E2 -6733.033} C_VEL
LIN {X 0,Y 481.696,Z 345.483,A -85,B 0,C 180,E1 -6735.638,E2 -6735.638} C_VEL
LIN {X 0,Y 481.758,Z 345.476,A -85,B 0,C 180,E1 -6738.215,E2 -6738.215} C_VEL
LIN {X 0,Y 481.77,Z 345.476,A -85,B 0,C 180,E1 -6741.611,E2 -6741.611} C_VEL
LIN {X 0,Y 481.783,Z 345.474,A -85,B 0,C 180,E1 -6743.534,E2 -6743.534} C_VEL
LIN {X 0,Y 484.209,Z 353.889,A -85,B 0,C 180,E1 -6743.959,E2 -6743.959} C_VEL
LIN {X 0,Y 483.91,Z 365.963,A -85,B 0,C 180,E1 -6744.583,E2 -6744.583} C_VEL
LIN {X 0,Y 483.522,Z 378.219,A -85,B 0,C 180,E1 -6745.414,E2 -6745.414} C_VEL
LIN {X 0,Y 483.084,Z 389.005,A -85,B 0,C 180,E1 -6746.35,E2 -6746.35} C_VEL
LIN {X 0,Y 482.626,Z 399.499,A -85,B 0,C 180,E1 -6747.496,E2 -6747.496} C_VEL
LIN {X 0,Y 482.297,Z 407.25,A -85,B 0,C 180,E1 -6748.538,E2 -6748.538} C_VEL
LIN {X 0,Y 481.939,Z 414.867,A -85,B 0,C 180,E1 -6749.791,E2 -6749.791} C_VEL
LIN {X 0,Y 481.576,Z 421.85,A -85,B 0,C 180,E1 -6751.254,E2 -6751.254} C_VEL
LIN {X 0,Y 481.455,Z 426.504,A -85,B 0,C 180,E1 -6752.509,E2 -6752.509} C_VEL
LIN {X 0,Y 481.33,Z 430.091,A -85,B 0,C 180,E1 -6753.767,E2 -6753.767} C_VEL
LIN {X 0,Y 481.207,Z 432.699,A -85,B 0,C 180,E1 -6755.027,E2 -6755.027} C_VEL
LIN {X 0,Y 481.227,Z 433.921,A -85,B 0,C 180,E1 -6755.867,E2 -6755.867} C_VEL
LIN {X 0,Y 481.204,Z 434.76,A -85,B 0,C 180,E1 -6756.709,E2 -6756.709} C_VEL
LIN {X 0,Y 481.173,Z 435.207,A -85,B 0,C 180,E1 -6758.398,E2 -6758.398} C_VEL
LIN {X 0,Y 481.152,Z 434.866,A -85,B 0,C 180,E1 -6759.245,E2 -6759.245} C_VEL
LIN {X 0,Y 481.145,Z 434.13,A -85,B 0,C 180,E1 -6760.094,E2 -6760.094} C_VEL
LIN {X 0,Y 481.249,Z 432.942,A -85,B 0,C 180,E1 -6760.943,E2 -6760.943} C_VEL
LIN {X 0,Y 481.338,Z 431.005,A -85,B 0,C 180,E1 -6761.965,E2 -6761.965} C_VEL
LIN {X 0,Y 481.47,Z 426.845,A -85,B 0,C 180,E1 -6763.506,E2 -6763.506} C_VEL
LIN {X 0,Y 481.691,Z 422.134,A -85,B 0,C 180,E1 -6764.792,E2 -6764.792} C_VEL
LIN {X 0,Y 481.931,Z 416.125,A -85,B 0,C 180,E1 -6766.085,E2 -6766.085} C_VEL
LIN {X 0,Y 482.266,Z 408.583,A -85,B 0,C 180,E1 -6767.382,E2 -6767.382} C_VEL
LIN {X 0,Y 482.657,Z 400.798,A -85,B 0,C 180,E1 -6768.463,E2 -6768.463} C_VEL
LIN {X 0,Y 482.983,Z 391.183,A -85,B 0,C 180,E1 -6769.552,E2 -6769.552} C_VEL
LIN {X 0,Y 483.435,Z 380.42,A -85,B 0,C 180,E1 -6770.531,E2 -6770.531} C_VEL
LIN {X 0,Y 483.862,Z 369.933,A -85,B 0,C 180,E1 -6771.291,E2 -6771.291} C_VEL
LIN {X 0,Y 484.165,Z 359.321,A -85,B 0,C 180,E1 -6771.901,E2 -6771.901} C_VEL
LIN {X 0,Y 484.101,Z 353.611,A -85,B 0,C 180,E1 -6772.176,E2 -6772.176} C_VEL
LIN {X 0,Y 481.683,Z 345.485,A -85,B 0,C 180,E1 -6772.604,E2 -6772.604} C_VEL
LIN {X 0,Y 481.703,Z 345.485,A -85,B 0,C 180,E1 -6775.956,E2 -6775.956} C_VEL
LIN {X 0,Y 481.702,Z 345.485,A -85,B 0,C 180,E1 -6778.781,E2 -6778.781} C_VEL
LIN {X 0,Y 481.659,Z 345.492,A -85,B 0,C 180,E1 -6782.189,E2 -6782.189} C_VEL
LIN {X 0,Y 481.69,Z 345.488,A -85,B 0,C 180,E1 -6784.681,E2 -6784.681} C_VEL
LIN {X 0,Y 481.655,Z 345.489,A -85,B 0,C 180,E1 -6788.006,E2 -6788.006} C_VEL
LIN {X 0,Y 481.663,Z 345.489,A -85,B 0,C 180,E1 -6791.04,E2 -6791.04} C_VEL
LIN {X 0,Y 481.659,Z 345.49,A -85,B 0,C 180,E1 -6794.359,E2 -6794.359} C_VEL
LIN {X 0,Y 481.643,Z 345.49,A -85,B 0,C 180,E1 -6796.851,E2 -6796.851} C_VEL
LIN {X 0,Y 481.692,Z 345.484,A -85,B 0,C 180,E1 -6800.061,E2 -6800.061} C_VEL
LIN {X 0,Y 481.629,Z 345.494,A -85,B 0,C 180,E1 -6803.253,E2 -6803.253} C_VEL
LIN {X 0,Y 481.708,Z 345.485,A -85,B 0,C 180,E1 -6806.329,E2 -6806.329} C_VEL
LIN {X 0,Y 481.657,Z 345.475,A -85,B 0,C 180,E1 -6809.415,E2 -6809.415} C_VEL
LIN {X 0,Y 481.701,Z 345.479,A -85,B 0,C 180,E1 -6812.168,E2 -6812.168} C_VEL
LIN {X 0,Y 481.717,Z 345.481,A -85,B 0,C 180,E1 -6814.969,E2 -6814.969} C_VEL
LIN {X 0,Y 481.649,Z 345.488,A -85,B 0,C 180,E1 -6817.704,E2 -6817.704} C_VEL
LIN {X 0,Y 481.706,Z 345.484,A -85,B 0,C 180,E1 -6820.393,E2 -6820.393} C_VEL
LIN {X 0,Y 481.69,Z 345.482,A -85,B 0,C 180,E1 -6823.034,E2 -6823.034} C_VEL
LIN {X 0,Y 481.692,Z 345.485,A -85,B 0,C 180,E1 -6825.639,E2 -6825.639} C_VEL
LIN {X 0,Y 481.796,Z 345.473,A -85,B 0,C 180,E1 -6828.216,E2 -6828.216} C_VEL
LIN {X 0,Y 481.761,Z 345.477,A -85,B 0,C 180,E1 -6831.611,E2 -6831.611} C_VEL
LIN {X 0,Y 481.814,Z 345.466,A -85,B 0,C 180,E1 -6834.139,E2 -6834.139} C_VEL
LIN {X 0,Y 481.926,Z 345.456,A -85,B 0,C 180,E1 -6837.492,E2 -6837.492} C_VEL
LIN {X 0,Y 481.938,Z 345.45,A -85,B 0,C 180,E1 -6840,E2 -6840} C_VEL
LIN {X 0,Y 481.925,Z 345.457,A -85,B 0,C 180,E1 -6842.507,E2 -6842.507} C_VEL
LIN {X 0,Y 481.814,Z 345.467,A -85,B 0,C 180,E1 -6845.86,E2 -6845.86} C_VEL
LIN {X 0,Y 481.76,Z 345.477,A -85,B 0,C 180,E1 -6848.388,E2 -6848.388} C_VEL
LIN {X 0,Y 481.747,Z 345.478,A -85,B 0,C 180,E1 -6851.785,E2 -6851.785} C_VEL
LIN {X 0,Y 481.739,Z 345.48,A -85,B 0,C 180,E1 -6855.224,E2 -6855.224} C_VEL
LIN {X 0,Y 481.709,Z 345.483,A -85,B 0,C 180,E1 -6858.722,E2 -6858.722} C_VEL
LIN {X 0,Y 481.643,Z 345.492,A -85,B 0,C 180,E1 -6861.395,E2 -6861.395} C_VEL
LIN {X 0,Y 481.674,Z 345.488,A -85,B 0,C 180,E1 -6864.113,E2 -6864.113} C_VEL
LIN {X 0,Y 481.749,Z 345.481,A -85,B 0,C 180,E1 -6867.141,E2 -6867.141} C_VEL
LIN {X 0,Y 481.685,Z 345.487,A -85,B 0,C 180,E1 -6869.741,E2 -6869.741} C_VEL
LIN {X 0,Y 481.671,Z 345.488,A -85,B 0,C 180,E1 -6872.674,E2 -6872.674} C_VEL
LIN {X 0,Y 481.641,Z 345.491,A -85,B 0,C 180,E1 -6875.709,E2 -6875.709} C_VEL
LIN {X 0,Y 481.718,Z 345.481,A -85,B 0,C 180,E1 -6879.355,E2 -6879.355} C_VEL
LIN {X 0,Y 481.672,Z 345.485,A -85,B 0,C 180,E1 -6882.158,E2 -6882.158} C_VEL
LIN {X 0,Y 481.658,Z 345.487,A -85,B 0,C 180,E1 -6884.458,E2 -6884.458} C_VEL
LIN {X 0,Y 481.688,Z 345.483,A -85,B 0,C 180,E1 -6886.846,E2 -6886.846} C_VEL
LIN {X 0,Y 481.716,Z 345.539,A -85,B 0,C 180,E1 -6890.064,E2 -6890.064} C_VEL
LIN {X 0,Y 483.773,Z 356.463,A -85,B 0,C 180,E1 -6893.443,E2 -6893.443} C_VEL
LIN {X 0,Y 483.821,Z 360.113,A -85,B 0,C 180,E1 -6894.477,E2 -6894.477} C_VEL
LIN {X 0,Y 483.112,Z 373.097,A -85,B 0,C 180,E1 -6897.972,E2 -6897.972} C_VEL
LIN {X 0,Y 482.683,Z 384.346,A -85,B 0,C 180,E1 -6900.882,E2 -6900.882} C_VEL
LIN {X 0,Y 482.324,Z 395.242,A -85,B 0,C 180,E1 -6903.615,E2 -6903.615} C_VEL
LIN {X 0,Y 481.985,Z 407.965,A -85,B 0,C 180,E1 -6906.726,E2 -6906.726} C_VEL
LIN {X 0,Y 481.688,Z 421.438,A -85,B 0,C 180,E1 -6909.949,E2 -6909.949} C_VEL
LIN {X 0,Y 481.459,Z 434.514,A -85,B 0,C 180,E1 -6913.026,E2 -6913.026} C_VEL
LIN {X 0,Y 481.352,Z 443.013,A -85,B 0,C 180,E1 -6915.008,E2 -6915.008} C_VEL
LIN {X 0,Y 482.875,Z 458.462,A -85,B 0,C 180,E1 -6915.433,E2 -6915.433} C_VEL
LIN {X 0,Y 483.602,Z 465.389,A -85,B 0,C 180,E1 -6915.697,E2 -6915.697} C_VEL
LIN {X 0,Y 483.231,Z 477.114,A -85,B 0,C 180,E1 -6916.223,E2 -6916.223} C_VEL
LIN {X 0,Y 482.758,Z 489.529,A -85,B 0,C 180,E1 -6916.96,E2 -6916.96} C_VEL
LIN {X 0,Y 482.379,Z 501.076,A -85,B 0,C 180,E1 -6917.841,E2 -6917.841} C_VEL
LIN {X 0,Y 481.924,Z 511.709,A -85,B 0,C 180,E1 -6918.859,E2 -6918.859} C_VEL
LIN {X 0,Y 481.56,Z 520.704,A -85,B 0,C 180,E1 -6919.914,E2 -6919.914} C_VEL
LIN {X 0,Y 481.284,Z 529.505,A -85,B 0,C 180,E1 -6921.181,E2 -6921.181} C_VEL
LIN {X 0,Y 481.157,Z 536.559,A -85,B 0,C 180,E1 -6922.447,E2 -6922.447} C_VEL
LIN {X 0,Y 481.061,Z 542.232,A -85,B 0,C 180,E1 -6923.713,E2 -6923.713} C_VEL
LIN {X 0,Y 480.961,Z 546.663,A -85,B 0,C 180,E1 -6924.971,E2 -6924.971} C_VEL
LIN {X 0,Y 481.045,Z 549.033,A -85,B 0,C 180,E1 -6925.811,E2 -6925.811} C_VEL
LIN {X 0,Y 481.039,Z 550.947,A -85,B 0,C 180,E1 -6926.65,E2 -6926.65} C_VEL
LIN {X 0,Y 480.986,Z 552.378,A -85,B 0,C 180,E1 -6927.488,E2 -6927.488} C_VEL
LIN {X 0,Y 480.945,Z 553.399,A -85,B 0,C 180,E1 -6928.326,E2 -6928.326} C_VEL
LIN {X 0,Y 480.924,Z 554.025,A -85,B 0,C 180,E1 -6929.163,E2 -6929.163} C_VEL
LIN {X 0,Y 480.928,Z 554.252,A -85,B 0,C 180,E1 -6930.001,E2 -6930.001} C_VEL
LIN {X 0,Y 480.923,Z 554.034,A -85,B 0,C 180,E1 -6930.838,E2 -6930.838} C_VEL
LIN {X 0,Y 480.944,Z 553.419,A -85,B 0,C 180,E1 -6931.675,E2 -6931.675} C_VEL
LIN {X 0,Y 480.984,Z 552.407,A -85,B 0,C 180,E1 -6932.513,E2 -6932.513} C_VEL
LIN {X 0,Y 481.038,Z 550.985,A -85,B 0,C 180,E1 -6933.351,E2 -6933.351} C_VEL
LIN {X 0,Y 481.009,Z 547.978,A -85,B 0,C 180,E1 -6934.61,E2 -6934.61} C_VEL
LIN {X 0,Y 481.089,Z 543.921,A -85,B 0,C 180,E1 -6935.87,E2 -6935.87} C_VEL
LIN {X 0,Y 481.112,Z 537.669,A -85,B 0,C 180,E1 -6937.344,E2 -6937.344} C_VEL
LIN {X 0,Y 481.286,Z 530.863,A -85,B 0,C 180,E1 -6938.609,E2 -6938.609} C_VEL
LIN {X 0,Y 481.5,Z 522.429,A -85,B 0,C 180,E1 -6939.876,E2 -6939.876} C_VEL
LIN {X 0,Y 481.858,Z 513.809,A -85,B 0,C 180,E1 -6940.931,E2 -6940.931} C_VEL
LIN {X 0,Y 482.265,Z 503.472,A -85,B 0,C 180,E1 -6941.96,E2 -6941.96} C_VEL
LIN {X 0,Y 482.64,Z 492.677,A -85,B 0,C 180,E1 -6942.831,E2 -6942.831} C_VEL
LIN {X 0,Y 483.086,Z 481.196,A -85,B 0,C 180,E1 -6943.568,E2 -6943.568} C_VEL
LIN {X 0,Y 483.497,Z 469.423,A -85,B 0,C 180,E1 -6944.146,E2 -6944.146} C_VEL
LIN {X 0,Y 483.459,Z 462.535,A -85,B 0,C 180,E1 -6944.416,E2 -6944.416} C_VEL
LIN {X 0,Y 482.223,Z 451.618,A -85,B 0,C 180,E1 -6944.777,E2 -6944.777} C_VEL
LIN {X 0,Y 481.356,Z 443.19,A -85,B 0,C 180,E1 -6944.994,E2 -6944.994} C_VEL
LIN {X 0,Y 481.553,Z 429.687,A -85,B 0,C 180,E1 -6948.143,E2 -6948.143} C_VEL
LIN {X 0,Y 481.796,Z 417.546,A -85,B 0,C 180,E1 -6951.001,E2 -6951.001} C_VEL
LIN {X 0,Y 482.074,Z 404.55,A -85,B 0,C 180,E1 -6954.093,E2 -6954.093} C_VEL
LIN {X 0,Y 482.435,Z 391.298,A -85,B 0,C 180,E1 -6957.298,E2 -6957.298} C_VEL
LIN {X 0,Y 482.832,Z 377.876,A -85,B 0,C 180,E1 -6960.628,E2 -6960.628} C_VEL
LIN {X 0,Y 483.2,Z 366.426,A -85,B 0,C 180,E1 -6963.553,E2 -6963.553} C_VEL
LIN {X 0,Y 483.634,Z 356.912,A -85,B 0,C 180,E1 -6966.054,E2 -6966.054} C_VEL
LIN {X 0,Y 482.477,Z 349.62,A -85,B 0,C 180,E1 -6968.132,E2 -6968.132} C_VEL
LIN {X 0,Y 481.718,Z 345.484,A -85,B 0,C 180,E1 -6969.354,E2 -6969.354} C_VEL
LIN {X 0,Y 481.658,Z 345.491,A -85,B 0,C 180,E1 -6972.16,E2 -6972.16} C_VEL
LIN {X 0,Y 481.664,Z 345.488,A -85,B 0,C 180,E1 -6975.543,E2 -6975.543} C_VEL
LIN {X 0,Y 481.661,Z 345.489,A -85,B 0,C 180,E1 -6978.959,E2 -6978.959} C_VEL
LIN {X 0,Y 481.66,Z 345.488,A -85,B 0,C 180,E1 -6981.993,E2 -6981.993} C_VEL
LIN {X 0,Y 481.693,Z 345.485,A -85,B 0,C 180,E1 -6985.318,E2 -6985.318} C_VEL
LIN {X 0,Y 481.652,Z 345.489,A -85,B 0,C 180,E1 -6988.312,E2 -6988.312} C_VEL
LIN {X 0,Y 481.705,Z 345.483,A -85,B 0,C 180,E1 -6991.219,E2 -6991.219} C_VEL
LIN {X 0,Y 481.706,Z 345.483,A -85,B 0,C 180,E1 -6994.043,E2 -6994.043} C_VEL
LIN {X 0,Y 481.679,Z 345.487,A -85,B 0,C 180,E1 -6996.812,E2 -6996.812} C_VEL
LIN {X 0,Y 481.701,Z 345.483,A -85,B 0,C 180,E1 -6999.503,E2 -6999.503} C_VEL
LIN {X 0,Y 481.7,Z 345.486,A -85,B 0,C 180,E1 -7002.158,E2 -7002.158} C_VEL
LIN {X 0,Y 481.748,Z 345.478,A -85,B 0,C 180,E1 -7004.776,E2 -7004.776} C_VEL
LIN {X 0,Y 481.756,Z 345.477,A -85,B 0,C 180,E1 -7008.215,E2 -7008.215} C_VEL
LIN {X 0,Y 481.767,Z 345.474,A -85,B 0,C 180,E1 -7011.612,E2 -7011.612} C_VEL
LIN {X 0,Y 481.822,Z 345.47,A -85,B 0,C 180,E1 -7014.14,E2 -7014.14} C_VEL
LIN {X 0,Y 481.932,Z 345.454,A -85,B 0,C 180,E1 -7017.493,E2 -7017.493} C_VEL
LIN {X 0,Y 481.912,Z 345.458,A -85,B 0,C 180,E1 -7020.836,E2 -7020.836} C_VEL
LIN {X 0,Y 481.933,Z 345.455,A -85,B 0,C 180,E1 -7022.508,E2 -7022.508} C_VEL
LIN {X 0,Y 481.821,Z 345.47,A -85,B 0,C 180,E1 -7025.861,E2 -7025.861} C_VEL
LIN {X 0,Y 481.77,Z 345.476,A -85,B 0,C 180,E1 -7028.388,E2 -7028.388} C_VEL
LIN {X 0,Y 481.757,Z 345.477,A -85,B 0,C 180,E1 -7031.785,E2 -7031.785} C_VEL
LIN {X 0,Y 481.749,Z 345.476,A -85,B 0,C 180,E1 -7035.224,E2 -7035.224} C_VEL
LIN {X 0,Y 481.719,Z 345.481,A -85,B 0,C 180,E1 -7038.722,E2 -7038.722} C_VEL
LIN {X 0,Y 481.652,Z 345.491,A -85,B 0,C 180,E1 -7041.395,E2 -7041.395} C_VEL
LIN {X 0,Y 481.684,Z 345.486,A -85,B 0,C 180,E1 -7044.113,E2 -7044.113} C_VEL
LIN {X 0,Y 481.753,Z 345.478,A -85,B 0,C 180,E1 -7047.139,E2 -7047.139} C_VEL
LIN {X 0,Y 481.685,Z 345.486,A -85,B 0,C 180,E1 -7049.741,E2 -7049.741} C_VEL
LIN {X 0,Y 481.679,Z 345.486,A -85,B 0,C 180,E1 -7052.674,E2 -7052.674} C_VEL
LIN {X 0,Y 481.643,Z 345.493,A -85,B 0,C 180,E1 -7055.709,E2 -7055.709} C_VEL
LIN {X 0,Y 481.678,Z 345.485,A -85,B 0,C 180,E1 -7058.859,E2 -7058.859} C_VEL
LIN {X 0,Y 481.659,Z 345.489,A -85,B 0,C 180,E1 -7061.913,E2 -7061.913} C_VEL
LIN {X 0,Y 481.666,Z 345.487,A -85,B 0,C 180,E1 -7064.457,E2 -7064.457} C_VEL
LIN {X 0,Y 481.655,Z 345.491,A -85,B 0,C 180,E1 -7067.839,E2 -7067.839} C_VEL
LIN {X 0,Y 481.686,Z 345.486,A -85,B 0,C 180,E1 -7070.651,E2 -7070.651} C_VEL
LIN {X 0,Y 481.628,Z 345.494,A -85,B 0,C 180,E1 -7073.377,E2 -7073.377} C_VEL
LIN {X 0,Y 481.717,Z 345.481,A -85,B 0,C 180,E1 -7076.33,E2 -7076.33} C_VEL
LIN {X 0,Y 481.657,Z 345.49,A -85,B 0,C 180,E1 -7079.417,E2 -7079.417} C_VEL
LIN {X 0,Y 481.706,Z 345.481,A -85,B 0,C 180,E1 -7082.168,E2 -7082.168} C_VEL
LIN {X 0,Y 481.725,Z 345.483,A -85,B 0,C 180,E1 -7084.97,E2 -7084.97} C_VEL
LIN {X 0,Y 481.642,Z 345.489,A -85,B 0,C 180,E1 -7087.981,E2 -7087.981} C_VEL
LIN {X 0,Y 480.975,Z 345.575,A -85,B 0,C 180,E1 -7088.679,E2 -7088.679} C_VEL
LIN {X 0,Y 478.149,Z 345.927,A -85,B 0,C 180,E1 -7089.813,E2 -7089.813} C_VEL
LIN {X 0,Y 475.765,Z 346.225,A -85,B 0,C 180,E1 -7090.727,E2 -7090.727} C_VEL
LIN {X 0,Y 474.744,Z 346.351,A -85,B 0,C 180,E1 -7091.433,E2 -7091.433} C_VEL
LIN {X 0,Y 474.661,Z 346.36,A -85,B 0,C 180,E1 -7091.672,E2 -7091.672} C_VEL
LIN {X 0,Y 474.707,Z 346.355,A -85,B 0,C 180,E1 -7094.544,E2 -7094.544} C_VEL
LIN {X 0,Y 474.711,Z 346.353,A -85,B 0,C 180,E1 -7098.037,E2 -7098.037} C_VEL
LIN {X 0,Y 474.735,Z 346.351,A -85,B 0,C 180,E1 -7101.486,E2 -7101.486} C_VEL
LIN {X 0,Y 474.737,Z 346.352,A -85,B 0,C 180,E1 -7103.331,E2 -7103.331} C_VEL
LIN {X 0,Y 477.343,Z 355.892,A -85,B 0,C 180,E1 -7103.819,E2 -7103.819} C_VEL
LIN {X 0,Y 476.996,Z 368.575,A -85,B 0,C 180,E1 -7104.504,E2 -7104.504} C_VEL
LIN {X 0,Y 476.637,Z 379.113,A -85,B 0,C 180,E1 -7105.242,E2 -7105.242} C_VEL
LIN {X 0,Y 476.171,Z 389.898,A -85,B 0,C 180,E1 -7106.191,E2 -7106.191} C_VEL
LIN {X 0,Y 475.745,Z 399.52,A -85,B 0,C 180,E1 -7107.248,E2 -7107.248} C_VEL
LIN {X 0,Y 475.315,Z 408.857,A -85,B 0,C 180,E1 -7108.517,E2 -7108.517} C_VEL
LIN {X 0,Y 474.924,Z 416.302,A -85,B 0,C 180,E1 -7109.787,E2 -7109.787} C_VEL
LIN {X 0,Y 474.56,Z 423.179,A -85,B 0,C 180,E1 -7111.272,E2 -7111.272} C_VEL
LIN {X 0,Y 474.439,Z 427.737,A -85,B 0,C 180,E1 -7112.546,E2 -7112.546} C_VEL
LIN {X 0,Y 474.312,Z 430.198,A -85,B 0,C 180,E1 -7113.397,E2 -7113.397} C_VEL
LIN {X 0,Y 474.172,Z 433.757,A -85,B 0,C 180,E1 -7115.101,E2 -7115.101} C_VEL
LIN {X 0,Y 474.197,Z 434.936,A -85,B 0,C 180,E1 -7115.954,E2 -7115.954} C_VEL
LIN {X 0,Y 474.18,Z 435.694,A -85,B 0,C 180,E1 -7116.809,E2 -7116.809} C_VEL
LIN {X 0,Y 474.148,Z 436.057,A -85,B 0,C 180,E1 -7118.523,E2 -7118.523} C_VEL
LIN {X 0,Y 474.122,Z 435.675,A -85,B 0,C 180,E1 -7119.384,E2 -7119.384} C_VEL
LIN {X 0,Y 474.115,Z 434.858,A -85,B 0,C 180,E1 -7120.246,E2 -7120.246} C_VEL
LIN {X 0,Y 474.229,Z 433.626,A -85,B 0,C 180,E1 -7121.107,E2 -7121.107} C_VEL
LIN {X 0,Y 474.336,Z 431.798,A -85,B 0,C 180,E1 -7122.069,E2 -7122.069} C_VEL
LIN {X 0,Y 474.434,Z 428.698,A -85,B 0,C 180,E1 -7123.273,E2 -7123.273} C_VEL
LIN {X 0,Y 474.616,Z 424.296,A -85,B 0,C 180,E1 -7124.579,E2 -7124.579} C_VEL
LIN {X 0,Y 474.919,Z 418.069,A -85,B 0,C 180,E1 -7126.004,E2 -7126.004} C_VEL
LIN {X 0,Y 475.284,Z 410.118,A -85,B 0,C 180,E1 -7127.423,E2 -7127.423} C_VEL
LIN {X 0,Y 475.713,Z 402.483,A -85,B 0,C 180,E1 -7128.519,E2 -7128.519} C_VEL
LIN {X 0,Y 476.1,Z 393.13,A -85,B 0,C 180,E1 -7129.622,E2 -7129.622} C_VEL
LIN {X 0,Y 476.529,Z 382.597,A -85,B 0,C 180,E1 -7130.616,E2 -7130.616} C_VEL
LIN {X 0,Y 476.952,Z 372.41,A -85,B 0,C 180,E1 -7131.388,E2 -7131.388} C_VEL
LIN {X 0,Y 477.331,Z 362.039,A -85,B 0,C 180,E1 -7132.015,E2 -7132.015} C_VEL
LIN {X 0,Y 477.4,Z 356.176,A -85,B 0,C 180,E1 -7132.311,E2 -7132.311} C_VEL
LIN {X 0,Y 474.653,Z 346.361,A -85,B 0,C 180,E1 -7132.844,E2 -7132.844} C_VEL
LIN {X 0,Y 474.673,Z 346.361,A -85,B 0,C 180,E1 -7135.427,E2 -7135.427} C_VEL
LIN {X 0,Y 474.648,Z 346.365,A -85,B 0,C 180,E1 -7138.282,E2 -7138.282} C_VEL
LIN {X 0,Y 474.601,Z 346.368,A -85,B 0,C 180,E1 -7141.217,E2 -7141.217} C_VEL
LIN {X 0,Y 474.632,Z 346.364,A -85,B 0,C 180,E1 -7144.24,E2 -7144.24} C_VEL
LIN {X 0,Y 474.591,Z 346.372,A -85,B 0,C 180,E1 -7147.383,E2 -7147.383} C_VEL
LIN {X 0,Y 474.628,Z 346.365,A -85,B 0,C 180,E1 -7149.647,E2 -7149.647} C_VEL
LIN {X 0,Y 474.635,Z 346.364,A -85,B 0,C 180,E1 -7152.931,E2 -7152.931} C_VEL
LIN {X 0,Y 474.609,Z 346.368,A -85,B 0,C 180,E1 -7155.894,E2 -7155.894} C_VEL
LIN {X 0,Y 474.641,Z 346.365,A -85,B 0,C 180,E1 -7159.038,E2 -7159.038} C_VEL
LIN {X 0,Y 474.619,Z 346.368,A -85,B 0,C 180,E1 -7161.702,E2 -7161.702} C_VEL
LIN {X 0,Y 474.63,Z 346.365,A -85,B 0,C 180,E1 -7164.726,E2 -7164.726} C_VEL
LIN {X 0,Y 474.637,Z 346.359,A -85,B 0,C 180,E1 -7167.787,E2 -7167.787} C_VEL
LIN {X 0,Y 474.631,Z 346.354,A -85,B 0,C 180,E1 -7170.882,E2 -7170.882} C_VEL
LIN {X 0,Y 474.665,Z 346.36,A -85,B 0,C 180,E1 -7173.628,E2 -7173.628} C_VEL
LIN {X 0,Y 474.633,Z 346.359,A -85,B 0,C 180,E1 -7176.641,E2 -7176.641} C_VEL
LIN {X 0,Y 474.655,Z 346.362,A -85,B 0,C 180,E1 -7180.089,E2 -7180.089} C_VEL
LIN {X 0,Y 474.649,Z 346.359,A -85,B 0,C 180,E1 -7182.774,E2 -7182.774} C_VEL
LIN {X 0,Y 474.65,Z 346.364,A -85,B 0,C 180,E1 -7185.421,E2 -7185.421} C_VEL
LIN {X 0,Y 474.739,Z 346.351,A -85,B 0,C 180,E1 -7188.038,E2 -7188.038} C_VEL
LIN {X 0,Y 474.727,Z 346.353,A -85,B 0,C 180,E1 -7191.486,E2 -7191.486} C_VEL
LIN {X 0,Y 474.777,Z 346.342,A -85,B 0,C 180,E1 -7194.052,E2 -7194.052} C_VEL
LIN {X 0,Y 474.892,Z 346.333,A -85,B 0,C 180,E1 -7197.455,E2 -7197.455} C_VEL
LIN {X 0,Y 474.874,Z 346.332,A -85,B 0,C 180,E1 -7200.848,E2 -7200.848} C_VEL
LIN {X 0,Y 474.892,Z 346.333,A -85,B 0,C 180,E1 -7202.544,E2 -7202.544} C_VEL
LIN {X 0,Y 474.777,Z 346.344,A -85,B 0,C 180,E1 -7205.947,E2 -7205.947} C_VEL
LIN {X 0,Y 474.725,Z 346.352,A -85,B 0,C 180,E1 -7208.513,E2 -7208.513} C_VEL
LIN {X 0,Y 474.7,Z 346.356,A -85,B 0,C 180,E1 -7211.962,E2 -7211.962} C_VEL
LIN {X 0,Y 474.696,Z 346.357,A -85,B 0,C 180,E1 -7215.456,E2 -7215.456} C_VEL
LIN {X 0,Y 474.662,Z 346.361,A -85,B 0,C 180,E1 -7219.01,E2 -7219.01} C_VEL
LIN {X 0,Y 474.587,Z 346.37,A -85,B 0,C 180,E1 -7221.729,E2 -7221.729} C_VEL
LIN {X 0,Y 474.656,Z 346.363,A -85,B 0,C 180,E1 -7224.493,E2 -7224.493} C_VEL
LIN {X 0,Y 474.695,Z 346.359,A -85,B 0,C 180,E1 -7227.339,E2 -7227.339} C_VEL
LIN {X 0,Y 474.607,Z 346.369,A -85,B 0,C 180,E1 -7230.812,E2 -7230.812} C_VEL
LIN {X 0,Y 474.635,Z 346.365,A -85,B 0,C 180,E1 -7233.984,E2 -7233.984} C_VEL
LIN {X 0,Y 474.576,Z 346.373,A -85,B 0,C 180,E1 -7236.901,E2 -7236.901} C_VEL
LIN {X 0,Y 474.653,Z 346.362,A -85,B 0,C 180,E1 -7239.652,E2 -7239.652} C_VEL
LIN {X 0,Y 474.65,Z 346.364,A -85,B 0,C 180,E1 -7242.93,E2 -7242.93} C_VEL
LIN {X 0,Y 474.616,Z 346.366,A -85,B 0,C 180,E1 -7245.897,E2 -7245.897} C_VEL
LIN {X 0,Y 474.645,Z 346.366,A -85,B 0,C 180,E1 -7249.038,E2 -7249.038} C_VEL
LIN {X 0,Y 474.686,Z 346.571,A -85,B 0,C 180,E1 -7249.802,E2 -7249.802} C_VEL
LIN {X 0,Y 476.504,Z 355.99,A -85,B 0,C 180,E1 -7252.793,E2 -7252.793} C_VEL
LIN {X 0,Y 476.945,Z 360.536,A -85,B 0,C 180,E1 -7254.14,E2 -7254.14} C_VEL
LIN {X 0,Y 476.252,Z 371.868,A -85,B 0,C 180,E1 -7257.261,E2 -7257.261} C_VEL
LIN {X 0,Y 475.756,Z 383.344,A -85,B 0,C 180,E1 -7260.302,E2 -7260.302} C_VEL
LIN {X 0,Y 475.294,Z 396.481,A -85,B 0,C 180,E1 -7263.667,E2 -7263.667} C_VEL
LIN {X 0,Y 474.948,Z 408.069,A -85,B 0,C 180,E1 -7266.555,E2 -7266.555} C_VEL
LIN {X 0,Y 474.654,Z 420.693,A -85,B 0,C 180,E1 -7269.638,E2 -7269.638} C_VEL
LIN {X 0,Y 474.394,Z 433.705,A -85,B 0,C 180,E1 -7272.766,E2 -7272.766} C_VEL
LIN {X 0,Y 474.266,Z 442.154,A -85,B 0,C 180,E1 -7274.778,E2 -7274.778} C_VEL
LIN {X 0,Y 475.755,Z 456.87,A -85,B 0,C 180,E1 -7275.183,E2 -7275.183} C_VEL
LIN {X 0,Y 476.648,Z 465.931,A -85,B 0,C 180,E1 -7275.539,E2 -7275.539} C_VEL
LIN {X 0,Y 476.201,Z 478.304,A -85,B 0,C 180,E1 -7276.124,E2 -7276.124} C_VEL
LIN {X 0,Y 475.722,Z 490.241,A -85,B 0,C 180,E1 -7276.872,E2 -7276.872} C_VEL
LIN {X 0,Y 475.361,Z 500.76,A -85,B 0,C 180,E1 -7277.71,E2 -7277.71} C_VEL
LIN {X 0,Y 474.892,Z 510.822,A -85,B 0,C 180,E1 -7278.692,E2 -7278.692} C_VEL
LIN {X 0,Y 474.508,Z 519.812,A -85,B 0,C 180,E1 -7279.763,E2 -7279.763} C_VEL
LIN {X 0,Y 474.227,Z 528.612,A -85,B 0,C 180,E1 -7281.049,E2 -7281.049} C_VEL
LIN {X 0,Y 474.077,Z 535.667,A -85,B 0,C 180,E1 -7282.333,E2 -7282.333} C_VEL
LIN {X 0,Y 473.997,Z 541.685,A -85,B 0,C 180,E1 -7283.706,E2 -7283.706} C_VEL
LIN {X 0,Y 473.899,Z 545.78,A -85,B 0,C 180,E1 -7284.896,E2 -7284.896} C_VEL
LIN {X 0,Y 473.987,Z 548.153,A -85,B 0,C 180,E1 -7285.749,E2 -7285.749} C_VEL
LIN {X 0,Y 473.992,Z 550.07,A -85,B 0,C 180,E1 -7286.6,E2 -7286.6} C_VEL
LIN {X 0,Y 473.932,Z 551.501,A -85,B 0,C 180,E1 -7287.451,E2 -7287.451} C_VEL
LIN {X 0,Y 473.895,Z 552.525,A -85,B 0,C 180,E1 -7288.301,E2 -7288.301} C_VEL
LIN {X 0,Y 473.877,Z 553.153,A -85,B 0,C 180,E1 -7289.151,E2 -7289.151} C_VEL
LIN {X 0,Y 473.882,Z 553.381,A -85,B 0,C 180,E1 -7290.001,E2 -7290.001} C_VEL
LIN {X 0,Y 473.875,Z 553.163,A -85,B 0,C 180,E1 -7290.85,E2 -7290.85} C_VEL
LIN {X 0,Y 473.893,Z 552.548,A -85,B 0,C 180,E1 -7291.7,E2 -7291.7} C_VEL
LIN {X 0,Y 473.929,Z 551.537,A -85,B 0,C 180,E1 -7292.55,E2 -7292.55} C_VEL
LIN {X 0,Y 473.991,Z 550.116,A -85,B 0,C 180,E1 -7293.401,E2 -7293.401} C_VEL
LIN {X 0,Y 473.932,Z 547.105,A -85,B 0,C 180,E1 -7294.679,E2 -7294.679} C_VEL
LIN {X 0,Y 474.004,Z 543.045,A -85,B 0,C 180,E1 -7295.958,E2 -7295.958} C_VEL
LIN {X 0,Y 474.043,Z 536.793,A -85,B 0,C 180,E1 -7297.454,E2 -7297.454} C_VEL
LIN {X 0,Y 474.186,Z 529.982,A -85,B 0,C 180,E1 -7298.739,E2 -7298.739} C_VEL
LIN {X 0,Y 474.454,Z 521.549,A -85,B 0,C 180,E1 -7300.024,E2 -7300.024} C_VEL
LIN {X 0,Y 474.846,Z 512.925,A -85,B 0,C 180,E1 -7301.094,E2 -7301.094} C_VEL
LIN {X 0,Y 475.261,Z 502.849,A -85,B 0,C 180,E1 -7302.114,E2 -7302.114} C_VEL
LIN {X 0,Y 475.668,Z 491.771,A -85,B 0,C 180,E1 -7303.022,E2 -7303.022} C_VEL
LIN {X 0,Y 476.126,Z 480.261,A -85,B 0,C 180,E1 -7303.77,E2 -7303.77} C_VEL
LIN {X 0,Y 476.586,Z 468.446,A -85,B 0,C 180,E1 -7304.355,E2 -7304.355} C_VEL
LIN {X 0,Y 476.407,Z 462.755,A -85,B 0,C 180,E1 -7304.589,E2 -7304.589} C_VEL
LIN {X 0,Y 475.132,Z 450.444,A -85,B 0,C 180,E1 -7305.003,E2 -7305.003} C_VEL
LIN {X 0,Y 474.289,Z 442.415,A -85,B 0,C 180,E1 -7305.195,E2 -7305.195} C_VEL
LIN {X 0,Y 474.464,Z 430.091,A -85,B 0,C 180,E1 -7308.124,E2 -7308.124} C_VEL
LIN {X 0,Y 474.734,Z 416.469,A -85,B 0,C 180,E1 -7311.387,E2 -7311.387} C_VEL
LIN {X 0,Y 475.041,Z 403.735,A -85,B 0,C 180,E1 -7314.472,E2 -7314.472} C_VEL
LIN {X 0,Y 475.46,Z 390.148,A -85,B 0,C 180,E1 -7317.822,E2 -7317.822} C_VEL
LIN {X 0,Y 475.841,Z 377.362,A -85,B 0,C 180,E1 -7321.058,E2 -7321.058} C_VEL
LIN {X 0,Y 476.325,Z 365.674,A -85,B 0,C 180,E1 -7324.103,E2 -7324.103} C_VEL
LIN {X 0,Y 476.678,Z 358.078,A -85,B 0,C 180,E1 -7326.14,E2 -7326.14} C_VEL
LIN {X 0,Y 475.375,Z 350.237,A -85,B 0,C 180,E1 -7328.412,E2 -7328.412} C_VEL
LIN {X 0,Y 474.671,Z 346.361,A -85,B 0,C 180,E1 -7329.581,E2 -7329.581} C_VEL
LIN {X 0,Y 474.64,Z 346.365,A -85,B 0,C 180,E1 -7332.932,E2 -7332.932} C_VEL
LIN {X 0,Y 474.614,Z 346.367,A -85,B 0,C 180,E1 -7335.896,E2 -7335.896} C_VEL
LIN {X 0,Y 474.632,Z 346.365,A -85,B 0,C 180,E1 -7339.041,E2 -7339.041} C_VEL
LIN {X 0,Y 474.615,Z 346.366,A -85,B 0,C 180,E1 -7341.704,E2 -7341.704} C_VEL
LIN {X 0,Y 474.629,Z 346.365,A -85,B 0,C 180,E1 -7344.726,E2 -7344.726} C_VEL
LIN {X 0,Y 474.642,Z 346.361,A -85,B 0,C 180,E1 -7347.788,E2 -7347.788} C_VEL
LIN {X 0,Y 474.629,Z 346.366,A -85,B 0,C 180,E1 -7350.885,E2 -7350.885} C_VEL
LIN {X 0,Y 474.666,Z 346.359,A -85,B 0,C 180,E1 -7353.629,E2 -7353.629} C_VEL
LIN {X 0,Y 474.641,Z 346.364,A -85,B 0,C 180,E1 -7356.642,E2 -7356.642} C_VEL
LIN {X 0,Y 474.659,Z 346.361,A -85,B 0,C 180,E1 -7360.09,E2 -7360.09} C_VEL
LIN {X 0,Y 474.647,Z 346.364,A -85,B 0,C 180,E1 -7362.774,E2 -7362.774} C_VEL
LIN {X 0,Y 474.654,Z 346.361,A -85,B 0,C 180,E1 -7365.421,E2 -7365.421} C_VEL
LIN {X 0,Y 474.71,Z 346.355,A -85,B 0,C 180,E1 -7368.038,E2 -7368.038} C_VEL
LIN {X 0,Y 474.732,Z 346.35,A -85,B 0,C 180,E1 -7371.487,E2 -7371.487} C_VEL
LIN {X 0,Y 474.785,Z 346.346,A -85,B 0,C 180,E1 -7374.053,E2 -7374.053} C_VEL
LIN {X 0,Y 474.898,Z 346.33,A -85,B 0,C 180,E1 -7377.456,E2 -7377.456} C_VEL
LIN {X 0,Y 474.918,Z 346.331,A -85,B 0,C 180,E1 -7380,E2 -7380} C_VEL
LIN {X 0,Y 474.899,Z 346.331,A -85,B 0,C 180,E1 -7382.545,E2 -7382.545} C_VEL
LIN {X 0,Y 474.784,Z 346.346,A -85,B 0,C 180,E1 -7385.948,E2 -7385.948} C_VEL
LIN {X 0,Y 474.735,Z 346.352,A -85,B 0,C 180,E1 -7388.514,E2 -7388.514} C_VEL
LIN {X 0,Y 474.711,Z 346.356,A -85,B 0,C 180,E1 -7391.963,E2 -7391.963} C_VEL
LIN {X 0,Y 474.707,Z 346.355,A -85,B 0,C 180,E1 -7395.456,E2 -7395.456} C_VEL
LIN {X 0,Y 474.671,Z 346.359,A -85,B 0,C 180,E1 -7399.01,E2 -7399.01} C_VEL
LIN {X 0,Y 474.595,Z 346.369,A -85,B 0,C 180,E1 -7401.729,E2 -7401.729} C_VEL
LIN {X 0,Y 474.666,Z 346.36,A -85,B 0,C 180,E1 -7404.493,E2 -7404.493} C_VEL
LIN {X 0,Y 474.687,Z 346.358,A -85,B 0,C 180,E1 -7407.334,E2 -7407.334} C_VEL
LIN {X 0,Y 474.611,Z 346.365,A -85,B 0,C 180,E1 -7410.81,E2 -7410.81} C_VEL
LIN {X 0,Y 474.644,Z 346.363,A -85,B 0,C 180,E1 -7413.984,E2 -7413.984} C_VEL
LIN {X 0,Y 474.578,Z 346.371,A -85,B 0,C 180,E1 -7416.899,E2 -7416.899} C_VEL
LIN {X 0,Y 474.635,Z 346.364,A -85,B 0,C 180,E1 -7419.648,E2 -7419.648} C_VEL
LIN {X 0,Y 474.621,Z 346.366,A -85,B 0,C 180,E1 -7422.934,E2 -7422.934} C_VEL
LIN {X 0,Y 474.616,Z 346.366,A -85,B 0,C 180,E1 -7425.895,E2 -7425.895} C_VEL
LIN {X 0,Y 474.635,Z 346.365,A -85,B 0,C 180,E1 -7429.041,E2 -7429.041} C_VEL
LIN {X 0,Y 474.614,Z 346.366,A -85,B 0,C 180,E1 -7431.704,E2 -7431.704} C_VEL
LIN {X 0,Y 474.629,Z 346.365,A -85,B 0,C 180,E1 -7434.725,E2 -7434.725} C_VEL
LIN {X 0,Y 474.643,Z 346.363,A -85,B 0,C 180,E1 -7437.788,E2 -7437.788} C_VEL
LIN {X 0,Y 474.63,Z 346.365,A -85,B 0,C 180,E1 -7440.885,E2 -7440.885} C_VEL
LIN {X 0,Y 474.668,Z 346.36,A -85,B 0,C 180,E1 -7443.628,E2 -7443.628} C_VEL
LIN {X 0,Y 474.642,Z 346.363,A -85,B 0,C 180,E1 -7446.641,E2 -7446.641} C_VEL
LIN {X 0,Y 474.662,Z 346.359,A -85,B 0,C 180,E1 -7450.089,E2 -7450.089} C_VEL
LIN {X 0,Y 474.661,Z 346.36,A -85,B 0,C 180,E1 -7451.672,E2 -7451.672} C_VEL
LIN {X 0,Y 473.998,Z 346.444,A -85,B 0,C 180,E1 -7452.381,E2 -7452.381} C_VEL
LIN {X 0,Y 471.147,Z 346.799,A -85,B 0,C 180,E1 -7453.533,E2 -7453.533} C_VEL
LIN {X 0,Y 468.732,Z 347.1,A -85,B 0,C 180,E1 -7454.461,E2 -7454.461} C_VEL
LIN {X 0,Y 467.691,Z 347.229,A -85,B 0,C 180,E1 -7455.178,E2 -7455.178} C_VEL
LIN {X 0,Y 467.604,Z 347.238,A -85,B 0,C 180,E1 -7455.421,E2 -7455.421} C_VEL
LIN {X 0,Y 467.66,Z 347.234,A -85,B 0,C 180,E1 -7458.733,E2 -7458.733} C_VEL
LIN {X 0,Y 467.688,Z 347.229,A -85,B 0,C 180,E1 -7461.357,E2 -7461.357} C_VEL
LIN {X 0,Y 467.678,Z 347.232,A -85,B 0,C 180,E1 -7463.122,E2 -7463.122} C_VEL
LIN {X 0,Y 470.446,Z 356.726,A -85,B 0,C 180,E1 -7463.62,E2 -7463.62} C_VEL
LIN {X 0,Y 470.129,Z 369.403,A -85,B 0,C 180,E1 -7464.316,E2 -7464.316} C_VEL
LIN {X 0,Y 469.753,Z 379.951,A -85,B 0,C 180,E1 -7465.064,E2 -7465.064} C_VEL
LIN {X 0,Y 469.261,Z 390.749,A -85,B 0,C 180,E1 -7466.027,E2 -7466.027} C_VEL
LIN {X 0,Y 468.761,Z 401.25,A -85,B 0,C 180,E1 -7467.206,E2 -7467.206} C_VEL
LIN {X 0,Y 468.378,Z 409.007,A -85,B 0,C 180,E1 -7468.28,E2 -7468.28} C_VEL
LIN {X 0,Y 467.977,Z 416.623,A -85,B 0,C 180,E1 -7469.569,E2 -7469.569} C_VEL
LIN {X 0,Y 467.651,Z 422.719,A -85,B 0,C 180,E1 -7470.86,E2 -7470.86} C_VEL
LIN {X 0,Y 467.441,Z 427.568,A -85,B 0,C 180,E1 -7472.153,E2 -7472.153} C_VEL
LIN {X 0,Y 467.264,Z 431.331,A -85,B 0,C 180,E1 -7473.449,E2 -7473.449} C_VEL
LIN {X 0,Y 467.139,Z 434.807,A -85,B 0,C 180,E1 -7475.178,E2 -7475.178} C_VEL
LIN {X 0,Y 467.132,Z 436.561,A -85,B 0,C 180,E1 -7476.793,E2 -7476.793} C_VEL
LIN {X 0,Y 467.114,Z 436.957,A -85,B 0,C 180,E1 -7477.782,E2 -7477.782} C_VEL
LIN {X 0,Y 467.102,Z 436.912,A -85,B 0,C 180,E1 -7478.653,E2 -7478.653} C_VEL
LIN {X 0,Y 467.074,Z 436.464,A -85,B 0,C 180,E1 -7479.527,E2 -7479.527} C_VEL
LIN {X 0,Y 467.217,Z 434.319,A -85,B 0,C 180,E1 -7481.276,E2 -7481.276} C_VEL
LIN {X 0,Y 467.345,Z 431.614,A -85,B 0,C 180,E1 -7482.594,E2 -7482.594} C_VEL
LIN {X 0,Y 467.501,Z 427.869,A -85,B 0,C 180,E1 -7483.917,E2 -7483.917} C_VEL
LIN {X 0,Y 467.814,Z 422.962,A -85,B 0,C 180,E1 -7485.242,E2 -7485.242} C_VEL
LIN {X 0,Y 468.099,Z 416.741,A -85,B 0,C 180,E1 -7486.574,E2 -7486.574} C_VEL
LIN {X 0,Y 468.469,Z 408.864,A -85,B 0,C 180,E1 -7487.911,E2 -7487.911} C_VEL
LIN {X 0,Y 468.986,Z 400.087,A -85,B 0,C 180,E1 -7489.106,E2 -7489.106} C_VEL
LIN {X 0,Y 469.368,Z 390.783,A -85,B 0,C 180,E1 -7490.144,E2 -7490.144} C_VEL
LIN {X 0,Y 469.821,Z 380.867,A -85,B 0,C 180,E1 -7491.039,E2 -7491.039} C_VEL
LIN {X 0,Y 470.259,Z 369.969,A -85,B 0,C 180,E1 -7491.823,E2 -7491.823} C_VEL
LIN {X 0,Y 470.598,Z 357.529,A -85,B 0,C 180,E1 -7492.516,E2 -7492.516} C_VEL
LIN {X 0,Y 467.612,Z 347.238,A -85,B 0,C 180,E1 -7493.08,E2 -7493.08} C_VEL
LIN {X 0,Y 467.613,Z 347.24,A -85,B 0,C 180,E1 -7495.839,E2 -7495.839} C_VEL
LIN {X 0,Y 467.578,Z 347.244,A -85,B 0,C 180,E1 -7498.749,E2 -7498.749} C_VEL
LIN {X 0,Y 467.585,Z 347.246,A -85,B 0,C 180,E1 -7501.739,E2 -7501.739} C_VEL
LIN {X 0,Y 467.565,Z 347.247,A -85,B 0,C 180,E1 -7504.832,E2 -7504.832} C_VEL
LIN {X 0,Y 467.565,Z 347.244,A -85,B 0,C 180,E1 -7508.044,E2 -7508.044} C_VEL
LIN {X 0,Y 467.582,Z 347.244,A -85,B 0,C 180,E1 -7511.277,E2 -7511.277} C_VEL
LIN {X 0,Y 467.567,Z 347.244,A -85,B 0,C 180,E1 -7513.822,E2 -7513.822} C_VEL
LIN {X 0,Y 467.556,Z 347.248,A -85,B 0,C 180,E1 -7516.255,E2 -7516.255} C_VEL
LIN {X 0,Y 467.584,Z 347.244,A -85,B 0,C 180,E1 -7518.721,E2 -7518.721} C_VEL
LIN {X 0,Y 467.577,Z 347.245,A -85,B 0,C 180,E1 -7521.406,E2 -7521.406} C_VEL
LIN {X 0,Y 467.562,Z 347.244,A -85,B 0,C 180,E1 -7524.259,E2 -7524.259} C_VEL
LIN {X 0,Y 467.581,Z 347.241,A -85,B 0,C 180,E1 -7527.32,E2 -7527.32} C_VEL
LIN {X 0,Y 467.577,Z 347.23,A -85,B 0,C 180,E1 -7530.665,E2 -7530.665} C_VEL
LIN {X 0,Y 467.626,Z 347.235,A -85,B 0,C 180,E1 -7533.2,E2 -7533.2} C_VEL
LIN {X 0,Y 467.59,Z 347.237,A -85,B 0,C 180,E1 -7536.467,E2 -7536.467} C_VEL
LIN {X 0,Y 467.622,Z 347.237,A -85,B 0,C 180,E1 -7539.777,E2 -7539.777} C_VEL
LIN {X 0,Y 467.607,Z 347.236,A -85,B 0,C 180,E1 -7542.506,E2 -7542.506} C_VEL
LIN {X 0,Y 467.607,Z 347.241,A -85,B 0,C 180,E1 -7545.196,E2 -7545.196} C_VEL
LIN {X 0,Y 467.682,Z 347.23,A -85,B 0,C 180,E1 -7547.855,E2 -7547.855} C_VEL
LIN {X 0,Y 467.68,Z 347.232,A -85,B 0,C 180,E1 -7551.357,E2 -7551.357} C_VEL
LIN {X 0,Y 467.741,Z 347.218,A -85,B 0,C 180,E1 -7553.962,E2 -7553.962} C_VEL
LIN {X 0,Y 467.858,Z 347.209,A -85,B 0,C 180,E1 -7557.417,E2 -7557.417} C_VEL
LIN {X 0,Y 467.88,Z 347.2,A -85,B 0,C 180,E1 -7560,E2 -7560} C_VEL
LIN {X 0,Y 467.857,Z 347.209,A -85,B 0,C 180,E1 -7562.583,E2 -7562.583} C_VEL
LIN {X 0,Y 467.741,Z 347.221,A -85,B 0,C 180,E1 -7566.037,E2 -7566.037} C_VEL
LIN {X 0,Y 467.678,Z 347.229,A -85,B 0,C 180,E1 -7568.643,E2 -7568.643} C_VEL
LIN {X 0,Y 467.652,Z 347.235,A -85,B 0,C 180,E1 -7572.145,E2 -7572.145} C_VEL
LIN {X 0,Y 467.635,Z 347.236,A -85,B 0,C 180,E1 -7575.695,E2 -7575.695} C_VEL
LIN {X 0,Y 467.614,Z 347.239,A -85,B 0,C 180,E1 -7578.765,E2 -7578.765} C_VEL
LIN {X 0,Y 467.577,Z 347.244,A -85,B 0,C 180,E1 -7581.269,E2 -7581.269} C_VEL
LIN {X 0,Y 467.57,Z 347.243,A -85,B 0,C 180,E1 -7583.943,E2 -7583.943} C_VEL
LIN {X 0,Y 467.624,Z 347.239,A -85,B 0,C 180,E1 -7586.8,E2 -7586.8} C_VEL
LIN {X 0,Y 467.584,Z 347.243,A -85,B 0,C 180,E1 -7589.736,E2 -7589.736} C_VEL
LIN {X 0,Y 467.581,Z 347.244,A -85,B 0,C 180,E1 -7592.759,E2 -7592.759} C_VEL
LIN {X 0,Y 467.555,Z 347.245,A -85,B 0,C 180,E1 -7595.89,E2 -7595.89} C_VEL
LIN {X 0,Y 467.617,Z 347.235,A -85,B 0,C 180,E1 -7599.141,E2 -7599.141} C_VEL
LIN {X 0,Y 467.616,Z 347.239,A -85,B 0,C 180,E1 -7602.572,E2 -7602.572} C_VEL
LIN {X 0,Y 467.573,Z 347.241,A -85,B 0,C 180,E1 -7606.177,E2 -7606.177} C_VEL
LIN {X 0,Y 467.605,Z 347.244,A -85,B 0,C 180,E1 -7609.172,E2 -7609.172} C_VEL
LIN {X 0,Y 467.648,Z 347.383,A -85,B 0,C 180,E1 -7609.461,E2 -7609.461} C_VEL
LIN {X 0,Y 469.68,Z 357.987,A -85,B 0,C 180,E1 -7612.886,E2 -7612.886} C_VEL
LIN {X 0,Y 470.09,Z 361.099,A -85,B 0,C 180,E1 -7613.835,E2 -7613.835} C_VEL
LIN {X 0,Y 469.313,Z 372.346,A -85,B 0,C 180,E1 -7616.993,E2 -7616.993} C_VEL
LIN {X 0,Y 468.809,Z 382.918,A -85,B 0,C 180,E1 -7619.855,E2 -7619.855} C_VEL
LIN {X 0,Y 468.304,Z 395.852,A -85,B 0,C 180,E1 -7623.243,E2 -7623.243} C_VEL
LIN {X 0,Y 467.913,Z 408.179,A -85,B 0,C 180,E1 -7626.379,E2 -7626.379} C_VEL
LIN {X 0,Y 467.545,Z 421.818,A -85,B 0,C 180,E1 -7629.774,E2 -7629.774} C_VEL
LIN {X 0,Y 467.294,Z 434.753,A -85,B 0,C 180,E1 -7632.947,E2 -7632.947} C_VEL
LIN {X 0,Y 467.176,Z 441.207,A -85,B 0,C 180,E1 -7634.513,E2 -7634.513} C_VEL
LIN {X 0,Y 468.794,Z 456.845,A -85,B 0,C 180,E1 -7634.972,E2 -7634.972} C_VEL
LIN {X 0,Y 469.715,Z 466.613,A -85,B 0,C 180,E1 -7635.376,E2 -7635.376} C_VEL
LIN {X 0,Y 469.303,Z 477.598,A -85,B 0,C 180,E1 -7635.916,E2 -7635.916} C_VEL
LIN {X 0,Y 468.772,Z 489.47,A -85,B 0,C 180,E1 -7636.674,E2 -7636.674} C_VEL
LIN {X 0,Y 468.35,Z 500.488,A -85,B 0,C 180,E1 -7637.572,E2 -7637.572} C_VEL
LIN {X 0,Y 467.845,Z 509.987,A -85,B 0,C 180,E1 -7638.52,E2 -7638.52} C_VEL
LIN {X 0,Y 467.471,Z 518.959,A -85,B 0,C 180,E1 -7639.607,E2 -7639.607} C_VEL
LIN {X 0,Y 467.176,Z 527.745,A -85,B 0,C 180,E1 -7640.912,E2 -7640.912} C_VEL
LIN {X 0,Y 467.009,Z 534.791,A -85,B 0,C 180,E1 -7642.217,E2 -7642.217} C_VEL
LIN {X 0,Y 466.91,Z 541.145,A -85,B 0,C 180,E1 -7643.699,E2 -7643.699} C_VEL
LIN {X 0,Y 466.885,Z 546.168,A -85,B 0,C 180,E1 -7645.252,E2 -7645.252} C_VEL
LIN {X 0,Y 466.947,Z 549.194,A -85,B 0,C 180,E1 -7646.549,E2 -7646.549} C_VEL
LIN {X 0,Y 466.878,Z 550.626,A -85,B 0,C 180,E1 -7647.412,E2 -7647.412} C_VEL
LIN {X 0,Y 466.845,Z 551.651,A -85,B 0,C 180,E1 -7648.275,E2 -7648.275} C_VEL
LIN {X 0,Y 466.829,Z 552.28,A -85,B 0,C 180,E1 -7649.138,E2 -7649.138} C_VEL
LIN {X 0,Y 466.836,Z 552.509,A -85,B 0,C 180,E1 -7650.001,E2 -7650.001} C_VEL
LIN {X 0,Y 466.827,Z 552.292,A -85,B 0,C 180,E1 -7650.863,E2 -7650.863} C_VEL
LIN {X 0,Y 466.842,Z 551.677,A -85,B 0,C 180,E1 -7651.726,E2 -7651.726} C_VEL
LIN {X 0,Y 466.875,Z 550.665,A -85,B 0,C 180,E1 -7652.589,E2 -7652.589} C_VEL
LIN {X 0,Y 466.946,Z 549.245,A -85,B 0,C 180,E1 -7653.452,E2 -7653.452} C_VEL
LIN {X 0,Y 466.862,Z 546.229,A -85,B 0,C 180,E1 -7654.75,E2 -7654.75} C_VEL
LIN {X 0,Y 466.927,Z 542.166,A -85,B 0,C 180,E1 -7656.049,E2 -7656.049} C_VEL
LIN {X 0,Y 466.981,Z 535.909,A -85,B 0,C 180,E1 -7657.568,E2 -7657.568} C_VEL
LIN {X 0,Y 467.113,Z 529.084,A -85,B 0,C 180,E1 -7658.872,E2 -7658.872} C_VEL
LIN {X 0,Y 467.412,Z 520.64,A -85,B 0,C 180,E1 -7660.177,E2 -7660.177} C_VEL
LIN {X 0,Y 467.795,Z 511.995,A -85,B 0,C 180,E1 -7661.263,E2 -7661.263} C_VEL
LIN {X 0,Y 468.25,Z 502.171,A -85,B 0,C 180,E1 -7662.273,E2 -7662.273} C_VEL
LIN {X 0,Y 468.706,Z 490.785,A -85,B 0,C 180,E1 -7663.219,E2 -7663.219} C_VEL
LIN {X 0,Y 469.204,Z 479.237,A -85,B 0,C 180,E1 -7663.977,E2 -7663.977} C_VEL
LIN {X 0,Y 469.641,Z 467.335,A -85,B 0,C 180,E1 -7664.572,E2 -7664.572} C_VEL
LIN {X 0,Y 469.163,Z 461.442,A -85,B 0,C 180,E1 -7664.823,E2 -7664.823} C_VEL
LIN {X 0,Y 467.874,Z 447.833,A -85,B 0,C 180,E1 -7665.269,E2 -7665.269} C_VEL
LIN {X 0,Y 467.178,Z 441.509,A -85,B 0,C 180,E1 -7665.432,E2 -7665.432} C_VEL
LIN {X 0,Y 467.387,Z 428.083,A -85,B 0,C 180,E1 -7668.68,E2 -7668.68} C_VEL
LIN {X 0,Y 467.685,Z 415.998,A -85,B 0,C 180,E1 -7671.631,E2 -7671.631} C_VEL
LIN {X 0,Y 467.972,Z 404.79,A -85,B 0,C 180,E1 -7674.394,E2 -7674.394} C_VEL
LIN {X 0,Y 468.408,Z 391.515,A -85,B 0,C 180,E1 -7677.719,E2 -7677.719} C_VEL
LIN {X 0,Y 468.829,Z 378.857,A -85,B 0,C 180,E1 -7680.975,E2 -7680.975} C_VEL
